LIN {X 0,Y 417.024,Z 629.46,A -85,B 0,C 180,E1 -10170,E2 -10170} C_VEL
LIN {X 0,Y 417.067,Z 628.857,A -85,B 0,C 180,E1 -10171.932,E2 -10171.932} C_VEL
LIN {X 0,Y 416.992,Z 627.097,A -85,B 0,C 180,E1 -10173.866,E2 -10173.866} C_VEL
LIN {X 0,Y 417.045,Z 624.162,A -85,B 0,C 180,E1 -10175.804,E2 -10175.804} C_VEL
LIN {X 0,Y 417.18,Z 619.979,A -85,B 0,C 180,E1 -10177.746,E2 -10177.746} C_VEL
LIN {X 0,Y 417.416,Z 614.438,A -85,B 0,C 180,E1 -10179.694,E2 -10179.694} C_VEL
LIN {X 0,Y 417.947,Z 607.397,A -85,B 0,C 180,E1 -10181.642,E2 -10181.642} C_VEL
LIN {X 0,Y 418.576,Z 598.635,A -85,B 0,C 180,E1 -10183.596,E2 -10183.596} C_VEL
LIN {X 0,Y 419.465,Z 589.337,A -85,B 0,C 180,E1 -10185.301,E2 -10185.301} C_VEL
LIN {X 0,Y 420.438,Z 579.892,A -85,B 0,C 180,E1 -10186.76,E2 -10186.76} C_VEL
LIN {X 0,Y 421.622,Z 568.231,A -85,B 0,C 180,E1 -10188.269,E2 -10188.269} C_VEL
LIN {X 0,Y 422.9,Z 555.169,A -85,B 0,C 180,E1 -10189.666,E2 -10189.666} C_VEL
LIN {X 0,Y 424.296,Z 541.374,A -85,B 0,C 180,E1 -10190.863,E2 -10190.863} C_VEL
LIN {X 0,Y 425.468,Z 527.829,A -85,B 0,C 180,E1 -10191.819,E2 -10191.819} C_VEL
LIN {X 0,Y 426.543,Z 513.678,A -85,B 0,C 180,E1 -10192.609,E2 -10192.609} C_VEL
LIN {X 0,Y 427.474,Z 498.647,A -85,B 0,C 180,E1 -10193.24,E2 -10193.24} C_VEL
LIN {X 0,Y 428.206,Z 483.459,A -85,B 0,C 180,E1 -10193.679,E2 -10193.679} C_VEL
LIN {X 0,Y 430.543,Z 350.818,A -85,B 0,C 180,E1 -10195.955,E2 -10195.955} C_VEL
LIN {X 0,Y 425.078,Z 321.561,A -85,B 0,C 180,E1 -10196.849,E2 -10196.849} C_VEL
LIN {X 0,Y 424.032,Z 316.253,A -85,B 0,C 180,E1 -10197.038,E2 -10197.038} C_VEL
LIN {X 0,Y 424.69,Z 307.553,A -85,B 0,C 180,E1 -10198.455,E2 -10198.455} C_VEL
LIN {X 0,Y 422.236,Z 296.355,A -85,B 0,C 180,E1 -10200.53,E2 -10200.53} C_VEL
LIN {X 0,Y 418.282,Z 281.009,A -85,B 0,C 180,E1 -10203.568,E2 -10203.568} C_VEL
LIN {X 0,Y 418.242,Z 281.01,A -85,B 0,C 180,E1 -10207.225,E2 -10207.225} C_VEL
LIN {X 0,Y 418.244,Z 281.002,A -85,B 0,C 180,E1 -10209.683,E2 -10209.683} C_VEL
LIN {X 0,Y 418.226,Z 281.014,A -85,B 0,C 180,E1 -10212.321,E2 -10212.321} C_VEL
LIN {X 0,Y 418.238,Z 281.01,A -85,B 0,C 180,E1 -10215.109,E2 -10215.109} C_VEL
LIN {X 0,Y 418.243,Z 281.007,A -85,B 0,C 180,E1 -10217.767,E2 -10217.767} C_VEL
LIN {X 0,Y 418.248,Z 281.012,A -85,B 0,C 180,E1 -10220.621,E2 -10220.621} C_VEL
LIN {X 0,Y 418.245,Z 281.012,A -85,B 0,C 180,E1 -10223.976,E2 -10223.976} C_VEL
LIN {X 0,Y 418.261,Z 281.003,A -85,B 0,C 180,E1 -10227.156,E2 -10227.156} C_VEL
LIN {X 0,Y 418.265,Z 281.003,A -85,B 0,C 180,E1 -10230.838,E2 -10230.838} C_VEL
LIN {X 0,Y 418.24,Z 281.008,A -85,B 0,C 180,E1 -10234.094,E2 -10234.094} C_VEL
LIN {X 0,Y 418.236,Z 281.004,A -85,B 0,C 180,E1 -10237.264,E2 -10237.264} C_VEL
LIN {X 0,Y 418.288,Z 281.002,A -85,B 0,C 180,E1 -10240.365,E2 -10240.365} C_VEL
LIN {X 0,Y 418.321,Z 281,A -85,B 0,C 180,E1 -10243.405,E2 -10243.405} C_VEL
LIN {X 0,Y 418.352,Z 280.995,A -85,B 0,C 180,E1 -10247,E2 -10247} C_VEL
LIN {X 0,Y 418.34,Z 281,A -85,B 0,C 180,E1 -10250.329,E2 -10250.329} C_VEL
LIN {X 0,Y 418.446,Z 280.978,A -85,B 0,C 180,E1 -10253.248,E2 -10253.248} C_VEL
LIN {X 0,Y 418.323,Z 281,A -85,B 0,C 180,E1 -10255.181,E2 -10255.181} C_VEL
LIN {X 0,Y 418.538,Z 280.974,A -85,B 0,C 180,E1 -10258.076,E2 -10258.076} C_VEL
LIN {X 0,Y 418.412,Z 280.986,A -85,B 0,C 180,E1 -10260.963,E2 -10260.963} C_VEL
LIN {X 0,Y 418.486,Z 280.977,A -85,B 0,C 180,E1 -10262.888,E2 -10262.888} C_VEL
LIN {X 0,Y 418.443,Z 280.98,A -85,B 0,C 180,E1 -10266.752,E2 -10266.752} C_VEL
LIN {X 0,Y 418.331,Z 280.999,A -85,B 0,C 180,E1 -10269.672,E2 -10269.672} C_VEL
LIN {X 0,Y 418.351,Z 280.996,A -85,B 0,C 180,E1 -10273,E2 -10273} C_VEL
LIN {X 0,Y 418.262,Z 281.007,A -85,B 0,C 180,E1 -10276.71,E2 -10276.71} C_VEL
LIN {X 0,Y 418.246,Z 281.012,A -85,B 0,C 180,E1 -10279.779,E2 -10279.779} C_VEL
LIN {X 0,Y 418.228,Z 281.007,A -85,B 0,C 180,E1 -10282.737,E2 -10282.737} C_VEL
LIN {X 0,Y 418.214,Z 281.01,A -85,B 0,C 180,E1 -10285.908,E2 -10285.908} C_VEL
LIN {X 0,Y 418.258,Z 280.995,A -85,B 0,C 180,E1 -10289.163,E2 -10289.163} C_VEL
LIN {X 0,Y 418.234,Z 281.009,A -85,B 0,C 180,E1 -10292.529,E2 -10292.529} C_VEL
LIN {X 0,Y 418.25,Z 281.01,A -85,B 0,C 180,E1 -10294.842,E2 -10294.842} C_VEL
LIN {X 0,Y 418.229,Z 281.008,A -85,B 0,C 180,E1 -10298.445,E2 -10298.445} C_VEL
LIN {X 0,Y 418.208,Z 281.015,A -85,B 0,C 180,E1 -10300.95,E2 -10300.95} C_VEL
LIN {X 0,Y 418.182,Z 281.017,A -85,B 0,C 180,E1 -10303.724,E2 -10303.724} C_VEL
LIN {X 0,Y 418.157,Z 281.018,A -85,B 0,C 180,E1 -10306.441,E2 -10306.441} C_VEL
LIN {X 0,Y 418.208,Z 281.018,A -85,B 0,C 180,E1 -10309.133,E2 -10309.133} C_VEL
LIN {X 0,Y 418.233,Z 281.007,A -85,B 0,C 180,E1 -10312.774,E2 -10312.774} C_VEL
LIN {X 0,Y 418.229,Z 281.009,A -85,B 0,C 180,E1 -10316.32,E2 -10316.32} C_VEL
LIN {X 0,Y 418.235,Z 281.015,A -85,B 0,C 180,E1 -10319.727,E2 -10319.727} C_VEL
LIN {X 0,Y 418.26,Z 281.079,A -85,B 0,C 180,E1 -10321.106,E2 -10321.106} C_VEL
LIN {X 0,Y 420.163,Z 288.83,A -85,B 0,C 180,E1 -10322.78,E2 -10322.78} C_VEL
LIN {X 0,Y 430.381,Z 312.246,A -85,B 0,C 180,E1 -10323.914,E2 -10323.914} C_VEL
LIN {X 0,Y 430.959,Z 315.076,A -85,B 0,C 180,E1 -10324.004,E2 -10324.004} C_VEL
LIN {X 0,Y 429.175,Z 418.752,A -85,B 0,C 180,E1 -10325.769,E2 -10325.769} C_VEL
LIN {X 0,Y 428.544,Z 454.243,A -85,B 0,C 180,E1 -10326.405,E2 -10326.405} C_VEL
LIN {X 0,Y 427.949,Z 469.526,A -85,B 0,C 180,E1 -10326.866,E2 -10326.866} C_VEL
LIN {X 0,Y 427.171,Z 484.377,A -85,B 0,C 180,E1 -10327.512,E2 -10327.512} C_VEL
LIN {X 0,Y 426.162,Z 498.888,A -85,B 0,C 180,E1 -10328.346,E2 -10328.346} C_VEL
LIN {X 0,Y 425.104,Z 512.127,A -85,B 0,C 180,E1 -10329.305,E2 -10329.305} C_VEL
LIN {X 0,Y 423.74,Z 525.582,A -85,B 0,C 180,E1 -10330.501,E2 -10330.501} C_VEL
LIN {X 0,Y 423.01,Z 533.114,A -85,B 0,C 180,E1 -10331.296,E2 -10331.296} C_VEL
LIN {X 0,Y 421.968,Z 537.683,A -85,B 0,C 180,E1 -10331.788,E2 -10331.788} C_VEL
LIN {X 0,Y 418.449,Z 544.934,A -85,B 0,C 180,E1 -10332.576,E2 -10332.576} C_VEL
LIN {X 0,Y 414.904,Z 551.847,A -85,B 0,C 180,E1 -10333.424,E2 -10333.424} C_VEL
LIN {X 0,Y 413.805,Z 555.759,A -85,B 0,C 180,E1 -10334.017,E2 -10334.017} C_VEL
LIN {X 0,Y 412.722,Z 565.22,A -85,B 0,C 180,E1 -10335.705,E2 -10335.705} C_VEL
LIN {X 0,Y 411.949,Z 573.28,A -85,B 0,C 180,E1 -10337.436,E2 -10337.436} C_VEL
LIN {X 0,Y 411.195,Z 579.932,A -85,B 0,C 180,E1 -10339.163,E2 -10339.163} C_VEL
LIN {X 0,Y 410.68,Z 586.087,A -85,B 0,C 180,E1 -10341.14,E2 -10341.14} C_VEL
LIN {X 0,Y 410.333,Z 591.474,A -85,B 0,C 180,E1 -10343.414,E2 -10343.414} C_VEL
LIN {X 0,Y 410.121,Z 594.319,A -85,B 0,C 180,E1 -10345.084,E2 -10345.084} C_VEL
LIN {X 0,Y 410.09,Z 596.618,A -85,B 0,C 180,E1 -10347.052,E2 -10347.052} C_VEL
LIN {X 0,Y 409.958,Z 597.797,A -85,B 0,C 180,E1 -10349.017,E2 -10349.017} C_VEL
LIN {X 0,Y 409.958,Z 597.814,A -85,B 0,C 180,E1 -10350.982,E2 -10350.982} C_VEL
LIN {X 0,Y 410.09,Z 596.699,A -85,B 0,C 180,E1 -10352.947,E2 -10352.947} C_VEL
LIN {X 0,Y 410.119,Z 594.463,A -85,B 0,C 180,E1 -10354.915,E2 -10354.915} C_VEL
LIN {X 0,Y 410.334,Z 591.042,A -85,B 0,C 180,E1 -10356.885,E2 -10356.885} C_VEL
LIN {X 0,Y 410.669,Z 586.356,A -85,B 0,C 180,E1 -10358.86,E2 -10358.86} C_VEL
LIN {X 0,Y 411.17,Z 580.283,A -85,B 0,C 180,E1 -10360.837,E2 -10360.837} C_VEL
LIN {X 0,Y 411.997,Z 572.627,A -85,B 0,C 180,E1 -10362.812,E2 -10362.812} C_VEL
LIN {X 0,Y 412.813,Z 564.465,A -85,B 0,C 180,E1 -10364.543,E2 -10364.543} C_VEL
LIN {X 0,Y 413.919,Z 554.624,A -85,B 0,C 180,E1 -10366.269,E2 -10366.269} C_VEL
LIN {X 0,Y 415.038,Z 544.529,A -85,B 0,C 180,E1 -10367.746,E2 -10367.746} C_VEL
LIN {X 0,Y 416.417,Z 532.505,A -85,B 0,C 180,E1 -10369.214,E2 -10369.214} C_VEL
LIN {X 0,Y 417.512,Z 521.723,A -85,B 0,C 180,E1 -10370.315,E2 -10370.315} C_VEL
LIN {X 0,Y 418.779,Z 508.898,A -85,B 0,C 180,E1 -10371.408,E2 -10371.408} C_VEL
LIN {X 0,Y 419.917,Z 494.827,A -85,B 0,C 180,E1 -10372.38,E2 -10372.38} C_VEL
LIN {X 0,Y 420.902,Z 480.644,A -85,B 0,C 180,E1 -10373.145,E2 -10373.145} C_VEL
LIN {X 0,Y 421.646,Z 465.905,A -85,B 0,C 180,E1 -10373.743,E2 -10373.743} C_VEL
LIN {X 0,Y 422.11,Z 451.888,A -85,B 0,C 180,E1 -10374.139,E2 -10374.139} C_VEL
LIN {X 0,Y 424.203,Z 342.239,A -85,B 0,C 180,E1 -10376.042,E2 -10376.042} C_VEL
LIN {X 0,Y 424.592,Z 315.602,A -85,B 0,C 180,E1 -10376.51,E2 -10376.51} C_VEL
LIN {X 0,Y 415.445,Z 294.516,A -85,B 0,C 180,E1 -10377.55,E2 -10377.55} C_VEL
LIN {X 0,Y 412.915,Z 288.768,A -85,B 0,C 180,E1 -10377.864,E2 -10377.864} C_VEL
LIN {X 0,Y 411.194,Z 281.894,A -85,B 0,C 180,E1 -10379.484,E2 -10379.484} C_VEL
LIN {X 0,Y 411.201,Z 281.889,A -85,B 0,C 180,E1 -10383.156,E2 -10383.156} C_VEL
LIN {X 0,Y 411.187,Z 281.888,A -85,B 0,C 180,E1 -10386.551,E2 -10386.551} C_VEL
LIN {X 0,Y 411.166,Z 281.892,A -85,B 0,C 180,E1 -10389.72,E2 -10389.72} C_VEL
LIN {X 0,Y 411.159,Z 281.884,A -85,B 0,C 180,E1 -10393.135,E2 -10393.135} C_VEL
LIN {X 0,Y 411.161,Z 281.892,A -85,B 0,C 180,E1 -10395.882,E2 -10395.882} C_VEL
LIN {X 0,Y 411.153,Z 281.891,A -85,B 0,C 180,E1 -10399.492,E2 -10399.492} C_VEL
LIN {X 0,Y 411.175,Z 281.889,A -85,B 0,C 180,E1 -10402.024,E2 -10402.024} C_VEL
LIN {X 0,Y 411.197,Z 281.882,A -85,B 0,C 180,E1 -10405.124,E2 -10405.124} C_VEL
LIN {X 0,Y 411.151,Z 281.893,A -85,B 0,C 180,E1 -10408.001,E2 -10408.001} C_VEL
LIN {X 0,Y 411.166,Z 281.89,A -85,B 0,C 180,E1 -10411.406,E2 -10411.406} C_VEL
LIN {X 0,Y 411.186,Z 281.89,A -85,B 0,C 180,E1 -10414.941,E2 -10414.941} C_VEL
LIN {X 0,Y 411.196,Z 281.885,A -85,B 0,C 180,E1 -10417.913,E2 -10417.913} C_VEL
LIN {X 0,Y 411.181,Z 281.883,A -85,B 0,C 180,E1 -10421.049,E2 -10421.049} C_VEL
LIN {X 0,Y 411.206,Z 281.89,A -85,B 0,C 180,E1 -10424.13,E2 -10424.13} C_VEL
LIN {X 0,Y 411.302,Z 281.872,A -85,B 0,C 180,E1 -10427.165,E2 -10427.165} C_VEL
LIN {X 0,Y 411.28,Z 281.875,A -85,B 0,C 180,E1 -10430.161,E2 -10430.161} C_VEL
LIN {X 0,Y 411.386,Z 281.863,A -85,B 0,C 180,E1 -10433.132,E2 -10433.132} C_VEL
LIN {X 0,Y 411.288,Z 281.871,A -85,B 0,C 180,E1 -10435.099,E2 -10435.099} C_VEL
LIN {X 0,Y 411.507,Z 281.851,A -85,B 0,C 180,E1 -10438.042,E2 -10438.042} C_VEL
LIN {X 0,Y 411.435,Z 281.849,A -85,B 0,C 180,E1 -10440.979,E2 -10440.979} C_VEL
LIN {X 0,Y 411.434,Z 281.857,A -85,B 0,C 180,E1 -10442.937,E2 -10442.937} C_VEL
LIN {X 0,Y 411.431,Z 281.854,A -85,B 0,C 180,E1 -10445.883,E2 -10445.883} C_VEL
LIN {X 0,Y 411.316,Z 281.872,A -85,B 0,C 180,E1 -10448.846,E2 -10448.846} C_VEL
LIN {X 0,Y 411.281,Z 281.875,A -85,B 0,C 180,E1 -10451.833,E2 -10451.833} C_VEL
LIN {X 0,Y 411.258,Z 281.874,A -85,B 0,C 180,E1 -10454.853,E2 -10454.853} C_VEL
LIN {X 0,Y 411.249,Z 281.886,A -85,B 0,C 180,E1 -10457.915,E2 -10457.915} C_VEL
LIN {X 0,Y 411.195,Z 281.888,A -85,B 0,C 180,E1 -10461.034,E2 -10461.034} C_VEL
LIN {X 0,Y 411.216,Z 281.869,A -85,B 0,C 180,E1 -10464.216,E2 -10464.216} C_VEL
LIN {X 0,Y 411.187,Z 281.885,A -85,B 0,C 180,E1 -10467.483,E2 -10467.483} C_VEL
LIN {X 0,Y 411.187,Z 281.88,A -85,B 0,C 180,E1 -10470.848,E2 -10470.848} C_VEL
LIN {X 0,Y 411.205,Z 281.888,A -85,B 0,C 180,E1 -10474.334,E2 -10474.334} C_VEL
LIN {X 0,Y 411.194,Z 281.879,A -85,B 0,C 180,E1 -10477.974,E2 -10477.974} C_VEL
LIN {X 0,Y 411.181,Z 281.889,A -85,B 0,C 180,E1 -10480.504,E2 -10480.504} C_VEL
LIN {X 0,Y 411.171,Z 281.892,A -85,B 0,C 180,E1 -10483.134,E2 -10483.134} C_VEL
LIN {X 0,Y 411.166,Z 281.894,A -85,B 0,C 180,E1 -10485.881,E2 -10485.881} C_VEL
LIN {X 0,Y 411.161,Z 281.888,A -85,B 0,C 180,E1 -10488.772,E2 -10488.772} C_VEL
LIN {X 0,Y 411.193,Z 281.89,A -85,B 0,C 180,E1 -10492.027,E2 -10492.027} C_VEL
LIN {X 0,Y 411.212,Z 281.887,A -85,B 0,C 180,E1 -10495.667,E2 -10495.667} C_VEL
LIN {X 0,Y 411.244,Z 282.008,A -85,B 0,C 180,E1 -10496.04,E2 -10496.04} C_VEL
LIN {X 0,Y 415.337,Z 297.864,A -85,B 0,C 180,E1 -10499.212,E2 -10499.212} C_VEL
LIN {X 0,Y 417.858,Z 308.784,A -85,B 0,C 180,E1 -10501.286,E2 -10501.286} C_VEL
LIN {X 0,Y 417.385,Z 316.068,A -85,B 0,C 180,E1 -10502.504,E2 -10502.504} C_VEL
LIN {X 0,Y 422.472,Z 342.049,A -85,B 0,C 180,E1 -10503.347,E2 -10503.347} C_VEL
LIN {X 0,Y 424.118,Z 352.168,A -85,B 0,C 180,E1 -10503.645,E2 -10503.645} C_VEL
LIN {X 0,Y 421.823,Z 479.15,A -85,B 0,C 180,E1 -10505.844,E2 -10505.844} C_VEL
LIN {X 0,Y 421.165,Z 494.946,A -85,B 0,C 180,E1 -10506.261,E2 -10506.261} C_VEL
LIN {X 0,Y 420.254,Z 509.586,A -85,B 0,C 180,E1 -10506.836,E2 -10506.836} C_VEL
LIN {X 0,Y 419.189,Z 523.691,A -85,B 0,C 180,E1 -10507.579,E2 -10507.579} C_VEL
LIN {X 0,Y 417.898,Z 538.017,A -85,B 0,C 180,E1 -10508.545,E2 -10508.545} C_VEL
LIN {X 0,Y 416.582,Z 551.066,A -85,B 0,C 180,E1 -10509.638,E2 -10509.638} C_VEL
LIN {X 0,Y 415.288,Z 563.121,A -85,B 0,C 180,E1 -10510.86,E2 -10510.86} C_VEL
LIN {X 0,Y 414.076,Z 574.294,A -85,B 0,C 180,E1 -10512.212,E2 -10512.212} C_VEL
LIN {X 0,Y 412.993,Z 584.581,A -85,B 0,C 180,E1 -10513.693,E2 -10513.693} C_VEL
LIN {X 0,Y 411.981,Z 594.643,A -85,B 0,C 180,E1 -10515.427,E2 -10515.427} C_VEL
LIN {X 0,Y 411.192,Z 603.004,A -85,B 0,C 180,E1 -10517.163,E2 -10517.163} C_VEL
LIN {X 0,Y 410.641,Z 610.868,A -85,B 0,C 180,E1 -10519.149,E2 -10519.149} C_VEL
LIN {X 0,Y 410.223,Z 617.126,A -85,B 0,C 180,E1 -10521.131,E2 -10521.131} C_VEL
LIN {X 0,Y 410.049,Z 621.972,A -85,B 0,C 180,E1 -10523.11,E2 -10523.11} C_VEL
LIN {X 0,Y 409.957,Z 625.523,A -85,B 0,C 180,E1 -10525.083,E2 -10525.083} C_VEL
LIN {X 0,Y 409.934,Z 627.86,A -85,B 0,C 180,E1 -10527.052,E2 -10527.052} C_VEL
LIN {X 0,Y 409.953,Z 629.036,A -85,B 0,C 180,E1 -10529.018,E2 -10529.018} C_VEL
LIN {X 0,Y 409.953,Z 629.034,A -85,B 0,C 180,E1 -10530.983,E2 -10530.983} C_VEL
LIN {X 0,Y 409.935,Z 627.851,A -85,B 0,C 180,E1 -10532.949,E2 -10532.949} C_VEL
LIN {X 0,Y 409.953,Z 625.51,A -85,B 0,C 180,E1 -10534.918,E2 -10534.918} C_VEL
LIN {X 0,Y 410.047,Z 621.961,A -85,B 0,C 180,E1 -10536.891,E2 -10536.891} C_VEL
LIN {X 0,Y 410.222,Z 617.114,A -85,B 0,C 180,E1 -10538.87,E2 -10538.87} C_VEL
LIN {X 0,Y 410.639,Z 610.843,A -85,B 0,C 180,E1 -10540.852,E2 -10540.852} C_VEL
LIN {X 0,Y 411.19,Z 602.971,A -85,B 0,C 180,E1 -10542.838,E2 -10542.838} C_VEL
LIN {X 0,Y 411.982,Z 594.608,A -85,B 0,C 180,E1 -10544.574,E2 -10544.574} C_VEL
LIN {X 0,Y 412.959,Z 584.537,A -85,B 0,C 180,E1 -10546.309,E2 -10546.309} C_VEL
LIN {X 0,Y 414.128,Z 574.249,A -85,B 0,C 180,E1 -10547.787,E2 -10547.787} C_VEL
LIN {X 0,Y 415.449,Z 561.994,A -85,B 0,C 180,E1 -10549.262,E2 -10549.262} C_VEL
LIN {X 0,Y 416.733,Z 549.7,A -85,B 0,C 180,E1 -10550.484,E2 -10550.484} C_VEL
LIN {X 0,Y 418.056,Z 536.328,A -85,B 0,C 180,E1 -10551.577,E2 -10551.577} C_VEL
LIN {X 0,Y 419.357,Z 521.576,A -85,B 0,C 180,E1 -10552.543,E2 -10552.543} C_VEL
LIN {X 0,Y 420.489,Z 506.139,A -85,B 0,C 180,E1 -10553.316,E2 -10553.316} C_VEL
LIN {X 0,Y 421.356,Z 491.063,A -85,B 0,C 180,E1 -10553.859,E2 -10553.859} C_VEL
LIN {X 0,Y 421.913,Z 475.757,A -85,B 0,C 180,E1 -10554.217,E2 -10554.217} C_VEL
LIN {X 0,Y 424.075,Z 351.155,A -85,B 0,C 180,E1 -10556.369,E2 -10556.369} C_VEL
LIN {X 0,Y 418.263,Z 320.609,A -85,B 0,C 180,E1 -10557.335,E2 -10557.335} C_VEL
LIN {X 0,Y 417.351,Z 316.082,A -85,B 0,C 180,E1 -10557.487,E2 -10557.487} C_VEL
LIN {X 0,Y 417.893,Z 309.811,A -85,B 0,C 180,E1 -10558.526,E2 -10558.526} C_VEL
LIN {X 0,Y 415.748,Z 299.421,A -85,B 0,C 180,E1 -10560.474,E2 -10560.474} C_VEL
LIN {X 0,Y 411.516,Z 283.155,A -85,B 0,C 180,E1 -10563.714,E2 -10563.714} C_VEL
LIN {X 0,Y 411.22,Z 281.889,A -85,B 0,C 180,E1 -10564,E2 -10564} C_VEL
LIN {X 0,Y 411.192,Z 281.892,A -85,B 0,C 180,E1 -10566.743,E2 -10566.743} C_VEL
LIN {X 0,Y 411.209,Z 281.878,A -85,B 0,C 180,E1 -10569.727,E2 -10569.727} C_VEL
LIN {X 0,Y 411.173,Z 281.89,A -85,B 0,C 180,E1 -10573.134,E2 -10573.134} C_VEL
LIN {X 0,Y 411.17,Z 281.887,A -85,B 0,C 180,E1 -10575.882,E2 -10575.882} C_VEL
LIN {X 0,Y 411.167,Z 281.893,A -85,B 0,C 180,E1 -10578.772,E2 -10578.772} C_VEL
LIN {X 0,Y 411.194,Z 281.889,A -85,B 0,C 180,E1 -10582.026,E2 -10582.026} C_VEL
LIN {X 0,Y 411.209,Z 281.883,A -85,B 0,C 180,E1 -10585.667,E2 -10585.667} C_VEL
LIN {X 0,Y 411.193,Z 281.885,A -85,B 0,C 180,E1 -10589.153,E2 -10589.153} C_VEL
LIN {X 0,Y 411.193,Z 281.887,A -85,B 0,C 180,E1 -10592.518,E2 -10592.518} C_VEL
LIN {X 0,Y 411.216,Z 281.886,A -85,B 0,C 180,E1 -10595.784,E2 -10595.784} C_VEL
LIN {X 0,Y 411.201,Z 281.886,A -85,B 0,C 180,E1 -10598.966,E2 -10598.966} C_VEL
LIN {X 0,Y 411.255,Z 281.882,A -85,B 0,C 180,E1 -10602.085,E2 -10602.085} C_VEL
LIN {X 0,Y 411.264,Z 281.874,A -85,B 0,C 180,E1 -10605.148,E2 -10605.148} C_VEL
LIN {X 0,Y 411.287,Z 281.874,A -85,B 0,C 180,E1 -10608.167,E2 -10608.167} C_VEL
LIN {X 0,Y 411.322,Z 281.872,A -85,B 0,C 180,E1 -10611.154,E2 -10611.154} C_VEL
LIN {X 0,Y 411.434,Z 281.861,A -85,B 0,C 180,E1 -10614.118,E2 -10614.118} C_VEL
LIN {X 0,Y 411.507,Z 281.849,A -85,B 0,C 180,E1 -10618.043,E2 -10618.043} C_VEL
LIN {X 0,Y 411.382,Z 281.861,A -85,B 0,C 180,E1 -10620.979,E2 -10620.979} C_VEL
LIN {X 0,Y 411.444,Z 281.854,A -85,B 0,C 180,E1 -10622.937,E2 -10622.937} C_VEL
LIN {X 0,Y 411.393,Z 281.859,A -85,B 0,C 180,E1 -10626.868,E2 -10626.868} C_VEL
LIN {X 0,Y 411.285,Z 281.874,A -85,B 0,C 180,E1 -10629.839,E2 -10629.839} C_VEL
LIN {X 0,Y 411.311,Z 281.874,A -85,B 0,C 180,E1 -10633.104,E2 -10633.104} C_VEL
LIN {X 0,Y 411.212,Z 281.885,A -85,B 0,C 180,E1 -10636.891,E2 -10636.891} C_VEL
LIN {X 0,Y 411.208,Z 281.888,A -85,B 0,C 180,E1 -10639.988,E2 -10639.988} C_VEL
LIN {X 0,Y 411.188,Z 281.885,A -85,B 0,C 180,E1 -10643.149,E2 -10643.149} C_VEL
LIN {X 0,Y 411.167,Z 281.885,A -85,B 0,C 180,E1 -10646.386,E2 -10646.386} C_VEL
LIN {X 0,Y 411.196,Z 281.883,A -85,B 0,C 180,E1 -10649.713,E2 -10649.713} C_VEL
LIN {X 0,Y 411.206,Z 281.886,A -85,B 0,C 180,E1 -10653.156,E2 -10653.156} C_VEL
LIN {X 0,Y 411.19,Z 281.885,A -85,B 0,C 180,E1 -10656.551,E2 -10656.551} C_VEL
LIN {X 0,Y 411.166,Z 281.893,A -85,B 0,C 180,E1 -10659.719,E2 -10659.719} C_VEL
LIN {X 0,Y 411.12,Z 281.9,A -85,B 0,C 180,E1 -10663.141,E2 -10663.141} C_VEL
LIN {X 0,Y 411.111,Z 281.896,A -85,B 0,C 180,E1 -10665.889,E2 -10665.889} C_VEL
LIN {X 0,Y 411.158,Z 281.895,A -85,B 0,C 180,E1 -10669.492,E2 -10669.492} C_VEL
LIN {X 0,Y 411.179,Z 281.888,A -85,B 0,C 180,E1 -10672.024,E2 -10672.024} C_VEL
LIN {X 0,Y 411.201,Z 281.887,A -85,B 0,C 180,E1 -10675.124,E2 -10675.124} C_VEL
LIN {X 0,Y 411.155,Z 281.891,A -85,B 0,C 180,E1 -10678.001,E2 -10678.001} C_VEL
LIN {X 0,Y 411.218,Z 281.932,A -85,B 0,C 180,E1 -10680.683,E2 -10680.683} C_VEL
LIN {X 0,Y 412.926,Z 288.883,A -85,B 0,C 180,E1 -10682.257,E2 -10682.257} C_VEL
LIN {X 0,Y 423.835,Z 313.789,A -85,B 0,C 180,E1 -10683.503,E2 -10683.503} C_VEL
LIN {X 0,Y 424.541,Z 315.615,A -85,B 0,C 180,E1 -10683.585,E2 -10683.585} C_VEL
LIN {X 0,Y 422.796,Z 417.26,A -85,B 0,C 180,E1 -10685.346,E2 -10685.346} C_VEL
LIN {X 0,Y 422.061,Z 454.53,A -85,B 0,C 180,E1 -10686.02,E2 -10686.02} C_VEL
LIN {X 0,Y 421.457,Z 469.531,A -85,B 0,C 180,E1 -10686.477,E2 -10686.477} C_VEL
LIN {X 0,Y 420.629,Z 484.849,A -85,B 0,C 180,E1 -10687.154,E2 -10687.154} C_VEL
LIN {X 0,Y 419.586,Z 499.164,A -85,B 0,C 180,E1 -10687.989,E2 -10687.989} C_VEL
LIN {X 0,Y 418.456,Z 512.403,A -85,B 0,C 180,E1 -10688.961,E2 -10688.961} C_VEL
LIN {X 0,Y 417.045,Z 525.857,A -85,B 0,C 180,E1 -10690.175,E2 -10690.175} C_VEL
LIN {X 0,Y 415.803,Z 538.049,A -85,B 0,C 180,E1 -10691.523,E2 -10691.523} C_VEL
LIN {X 0,Y 414.582,Z 549.15,A -85,B 0,C 180,E1 -10692.996,E2 -10692.996} C_VEL
LIN {X 0,Y 413.805,Z 555.759,A -85,B 0,C 180,E1 -10694.017,E2 -10694.017} C_VEL
LIN {X 0,Y 412.723,Z 559.602,A -85,B 0,C 180,E1 -10694.631,E2 -10694.631} C_VEL
LIN {X 0,Y 406.401,Z 570.041,A -85,B 0,C 180,E1 -10696.448,E2 -10696.448} C_VEL
LIN {X 0,Y 405.096,Z 573.179,A -85,B 0,C 180,E1 -10697.13,E2 -10697.13} C_VEL
LIN {X 0,Y 404.938,Z 574.161,A -85,B 0,C 180,E1 -10697.37,E2 -10697.37} C_VEL
LIN {X 0,Y 404.046,Z 581.873,A -85,B 0,C 180,E1 -10699.476,E2 -10699.476} C_VEL
LIN {X 0,Y 403.538,Z 587.676,A -85,B 0,C 180,E1 -10701.486,E2 -10701.486} C_VEL
LIN {X 0,Y 403.271,Z 591.946,A -85,B 0,C 180,E1 -10703.398,E2 -10703.398} C_VEL
LIN {X 0,Y 403.06,Z 594.589,A -85,B 0,C 180,E1 -10704.998,E2 -10704.998} C_VEL
LIN {X 0,Y 402.992,Z 596.889,A -85,B 0,C 180,E1 -10707.001,E2 -10707.001} C_VEL
LIN {X 0,Y 402.884,Z 598.067,A -85,B 0,C 180,E1 -10709,E2 -10709} C_VEL
LIN {X 0,Y 402.884,Z 598.083,A -85,B 0,C 180,E1 -10710.999,E2 -10710.999} C_VEL
LIN {X 0,Y 402.992,Z 596.969,A -85,B 0,C 180,E1 -10712.999,E2 -10712.999} C_VEL
LIN {X 0,Y 403.058,Z 594.733,A -85,B 0,C 180,E1 -10715.001,E2 -10715.001} C_VEL
LIN {X 0,Y 403.272,Z 591.312,A -85,B 0,C 180,E1 -10717.007,E2 -10717.007} C_VEL
LIN {X 0,Y 403.649,Z 586.626,A -85,B 0,C 180,E1 -10719.015,E2 -10719.015} C_VEL
LIN {X 0,Y 404.164,Z 580.553,A -85,B 0,C 180,E1 -10721.027,E2 -10721.027} C_VEL
LIN {X 0,Y 405.048,Z 572.897,A -85,B 0,C 180,E1 -10723.036,E2 -10723.036} C_VEL
LIN {X 0,Y 405.91,Z 564.734,A -85,B 0,C 180,E1 -10724.796,E2 -10724.796} C_VEL
LIN {X 0,Y 407.094,Z 554.892,A -85,B 0,C 180,E1 -10726.55,E2 -10726.55} C_VEL
LIN {X 0,Y 408.256,Z 544.797,A -85,B 0,C 180,E1 -10728.051,E2 -10728.051} C_VEL
LIN {X 0,Y 409.719,Z 532.772,A -85,B 0,C 180,E1 -10729.54,E2 -10729.54} C_VEL
LIN {X 0,Y 410.875,Z 521.988,A -85,B 0,C 180,E1 -10730.658,E2 -10730.658} C_VEL
LIN {X 0,Y 412.174,Z 509.162,A -85,B 0,C 180,E1 -10731.768,E2 -10731.768} C_VEL
LIN {X 0,Y 413.366,Z 495.09,A -85,B 0,C 180,E1 -10732.755,E2 -10732.755} C_VEL
LIN {X 0,Y 414.421,Z 480.226,A -85,B 0,C 180,E1 -10733.564,E2 -10733.564} C_VEL
LIN {X 0,Y 415.198,Z 465.249,A -85,B 0,C 180,E1 -10734.168,E2 -10734.168} C_VEL
LIN {X 0,Y 415.755,Z 450.631,A -85,B 0,C 180,E1 -10734.565,E2 -10734.565} C_VEL
LIN {X 0,Y 417.913,Z 337.717,A -85,B 0,C 180,E1 -10736.554,E2 -10736.554} C_VEL
LIN {X 0,Y 418.174,Z 317.36,A -85,B 0,C 180,E1 -10736.921,E2 -10736.921} C_VEL
LIN {X 0,Y 408.769,Z 295.62,A -85,B 0,C 180,E1 -10738.023,E2 -10738.023} C_VEL
LIN {X 0,Y 405.704,Z 288.989,A -85,B 0,C 180,E1 -10738.42,E2 -10738.42} C_VEL
LIN {X 0,Y 404.15,Z 282.773,A -85,B 0,C 180,E1 -10739.895,E2 -10739.895} C_VEL
LIN {X 0,Y 404.165,Z 282.766,A -85,B 0,C 180,E1 -10743.418,E2 -10743.418} C_VEL
LIN {X 0,Y 404.132,Z 282.765,A -85,B 0,C 180,E1 -10746.247,E2 -10746.247} C_VEL
LIN {X 0,Y 404.131,Z 282.772,A -85,B 0,C 180,E1 -10748.759,E2 -10748.759} C_VEL
LIN {X 0,Y 404.103,Z 282.771,A -85,B 0,C 180,E1 -10751.596,E2 -10751.596} C_VEL
LIN {X 0,Y 404.141,Z 282.764,A -85,B 0,C 180,E1 -10754.521,E2 -10754.521} C_VEL
LIN {X 0,Y 404.117,Z 282.756,A -85,B 0,C 180,E1 -10757.293,E2 -10757.293} C_VEL
LIN {X 0,Y 404.131,Z 282.766,A -85,B 0,C 180,E1 -10759.951,E2 -10759.951} C_VEL
LIN {X 0,Y 404.127,Z 282.749,A -85,B 0,C 180,E1 -10763.126,E2 -10763.126} C_VEL
LIN {X 0,Y 404.133,Z 282.766,A -85,B 0,C 180,E1 -10766.187,E2 -10766.187} C_VEL
LIN {X 0,Y 404.137,Z 282.765,A -85,B 0,C 180,E1 -10769.714,E2 -10769.714} C_VEL
LIN {X 0,Y 404.1,Z 282.771,A -85,B 0,C 180,E1 -10773.116,E2 -10773.116} C_VEL
LIN {X 0,Y 404.144,Z 282.764,A -85,B 0,C 180,E1 -10776.424,E2 -10776.424} C_VEL
LIN {X 0,Y 404.148,Z 282.766,A -85,B 0,C 180,E1 -10779.89,E2 -10779.89} C_VEL
LIN {X 0,Y 404.153,Z 282.766,A -85,B 0,C 180,E1 -10783.022,E2 -10783.022} C_VEL
LIN {X 0,Y 404.282,Z 282.748,A -85,B 0,C 180,E1 -10786.939,E2 -10786.939} C_VEL
LIN {X 0,Y 404.247,Z 282.753,A -85,B 0,C 180,E1 -10789.988,E2 -10789.988} C_VEL
LIN {X 0,Y 404.337,Z 282.742,A -85,B 0,C 180,E1 -10793.011,E2 -10793.011} C_VEL
LIN {X 0,Y 404.258,Z 282.746,A -85,B 0,C 180,E1 -10795.013,E2 -10795.013} C_VEL
LIN {X 0,Y 404.476,Z 282.726,A -85,B 0,C 180,E1 -10798.008,E2 -10798.008} C_VEL
LIN {X 0,Y 404.4,Z 282.725,A -85,B 0,C 180,E1 -10800.996,E2 -10800.996} C_VEL
LIN {X 0,Y 404.393,Z 282.734,A -85,B 0,C 180,E1 -10802.988,E2 -10802.988} C_VEL
LIN {X 0,Y 404.379,Z 282.732,A -85,B 0,C 180,E1 -10805.985,E2 -10805.985} C_VEL
LIN {X 0,Y 404.263,Z 282.75,A -85,B 0,C 180,E1 -10809.002,E2 -10809.002} C_VEL
LIN {X 0,Y 404.254,Z 282.753,A -85,B 0,C 180,E1 -10812.041,E2 -10812.041} C_VEL
LIN {X 0,Y 404.204,Z 282.752,A -85,B 0,C 180,E1 -10815.118,E2 -10815.118} C_VEL
LIN {X 0,Y 404.206,Z 282.759,A -85,B 0,C 180,E1 -10818.238,E2 -10818.238} C_VEL
LIN {X 0,Y 404.137,Z 282.769,A -85,B 0,C 180,E1 -10821.419,E2 -10821.419} C_VEL
LIN {X 0,Y 404.165,Z 282.744,A -85,B 0,C 180,E1 -10824.666,E2 -10824.666} C_VEL
LIN {X 0,Y 404.129,Z 282.771,A -85,B 0,C 180,E1 -10828.005,E2 -10828.005} C_VEL
LIN {X 0,Y 404.142,Z 282.76,A -85,B 0,C 180,E1 -10830.285,E2 -10830.285} C_VEL
LIN {X 0,Y 404.143,Z 282.764,A -85,B 0,C 180,E1 -10833.812,E2 -10833.812} C_VEL
LIN {X 0,Y 404.135,Z 282.759,A -85,B 0,C 180,E1 -10836.875,E2 -10836.875} C_VEL
LIN {X 0,Y 404.146,Z 282.768,A -85,B 0,C 180,E1 -10840.08,E2 -10840.08} C_VEL
LIN {X 0,Y 404.151,Z 282.766,A -85,B 0,C 180,E1 -10843.084,E2 -10843.084} C_VEL
LIN {X 0,Y 404.146,Z 282.767,A -85,B 0,C 180,E1 -10845.926,E2 -10845.926} C_VEL
LIN {X 0,Y 404.116,Z 282.766,A -85,B 0,C 180,E1 -10848.635,E2 -10848.635} C_VEL
LIN {X 0,Y 404.152,Z 282.767,A -85,B 0,C 180,E1 -10851.492,E2 -10851.492} C_VEL
LIN {X 0,Y 404.162,Z 282.769,A -85,B 0,C 180,E1 -10855.286,E2 -10855.286} C_VEL
LIN {X 0,Y 404.2,Z 282.924,A -85,B 0,C 180,E1 -10855.592,E2 -10855.592} C_VEL
LIN {X 0,Y 408.033,Z 297.686,A -85,B 0,C 180,E1 -10858.621,E2 -10858.621} C_VEL
LIN {X 0,Y 410.922,Z 309.971,A -85,B 0,C 180,E1 -10861.014,E2 -10861.014} C_VEL
LIN {X 0,Y 410.924,Z 313.697,A -85,B 0,C 180,E1 -10861.666,E2 -10861.666} C_VEL
LIN {X 0,Y 410.734,Z 315.723,A -85,B 0,C 180,E1 -10862.007,E2 -10862.007} C_VEL
LIN {X 0,Y 415.04,Z 337.414,A -85,B 0,C 180,E1 -10862.748,E2 -10862.748} C_VEL
LIN {X 0,Y 417.76,Z 353.1,A -85,B 0,C 180,E1 -10863.234,E2 -10863.234} C_VEL
LIN {X 0,Y 415.343,Z 478.895,A -85,B 0,C 180,E1 -10865.442,E2 -10865.442} C_VEL
LIN {X 0,Y 414.659,Z 494.685,A -85,B 0,C 180,E1 -10865.865,E2 -10865.865} C_VEL
LIN {X 0,Y 413.659,Z 510.084,A -85,B 0,C 180,E1 -10866.483,E2 -10866.483} C_VEL
LIN {X 0,Y 412.619,Z 523.426,A -85,B 0,C 180,E1 -10867.202,E2 -10867.202} C_VEL
LIN {X 0,Y 411.259,Z 537.749,A -85,B 0,C 180,E1 -10868.181,E2 -10868.181} C_VEL
LIN {X 0,Y 409.879,Z 550.797,A -85,B 0,C 180,E1 -10869.29,E2 -10869.29} C_VEL
LIN {X 0,Y 408.392,Z 563.927,A -85,B 0,C 180,E1 -10870.654,E2 -10870.654} C_VEL
LIN {X 0,Y 407.06,Z 575.819,A -85,B 0,C 180,E1 -10872.155,E2 -10872.155} C_VEL
LIN {X 0,Y 405.926,Z 585.832,A -85,B 0,C 180,E1 -10873.66,E2 -10873.66} C_VEL
LIN {X 0,Y 404.905,Z 595.636,A -85,B 0,C 180,E1 -10875.424,E2 -10875.424} C_VEL
LIN {X 0,Y 404.131,Z 603.823,A -85,B 0,C 180,E1 -10877.19,E2 -10877.19} C_VEL
LIN {X 0,Y 403.594,Z 610.596,A -85,B 0,C 180,E1 -10878.957,E2 -10878.957} C_VEL
LIN {X 0,Y 403.151,Z 616.854,A -85,B 0,C 180,E1 -10880.974,E2 -10880.974} C_VEL
LIN {X 0,Y 402.97,Z 621.701,A -85,B 0,C 180,E1 -10882.988,E2 -10882.988} C_VEL
LIN {X 0,Y 402.87,Z 625.252,A -85,B 0,C 180,E1 -10884.997,E2 -10884.997} C_VEL
LIN {X 0,Y 402.833,Z 627.589,A -85,B 0,C 180,E1 -10887,E2 -10887} C_VEL
LIN {X 0,Y 402.879,Z 628.766,A -85,B 0,C 180,E1 -10889.001,E2 -10889.001} C_VEL
LIN {X 0,Y 402.879,Z 628.765,A -85,B 0,C 180,E1 -10891,E2 -10891} C_VEL
LIN {X 0,Y 402.833,Z 627.58,A -85,B 0,C 180,E1 -10893.001,E2 -10893.001} C_VEL
LIN {X 0,Y 402.867,Z 625.239,A -85,B 0,C 180,E1 -10895.004,E2 -10895.004} C_VEL
LIN {X 0,Y 402.968,Z 621.689,A -85,B 0,C 180,E1 -10897.013,E2 -10897.013} C_VEL
LIN {X 0,Y 403.149,Z 616.84,A -85,B 0,C 180,E1 -10899.027,E2 -10899.027} C_VEL
LIN {X 0,Y 403.591,Z 610.569,A -85,B 0,C 180,E1 -10901.044,E2 -10901.044} C_VEL
LIN {X 0,Y 404.159,Z 602.694,A -85,B 0,C 180,E1 -10903.066,E2 -10903.066} C_VEL
LIN {X 0,Y 405.023,Z 594.332,A -85,B 0,C 180,E1 -10904.83,E2 -10904.83} C_VEL
LIN {X 0,Y 406.094,Z 584.262,A -85,B 0,C 180,E1 -10906.593,E2 -10906.593} C_VEL
LIN {X 0,Y 407.285,Z 573.972,A -85,B 0,C 180,E1 -10908.096,E2 -10908.096} C_VEL
LIN {X 0,Y 408.696,Z 561.718,A -85,B 0,C 180,E1 -10909.593,E2 -10909.593} C_VEL
LIN {X 0,Y 410.191,Z 548.082,A -85,B 0,C 180,E1 -10910.957,E2 -10910.957} C_VEL
LIN {X 0,Y 411.563,Z 534.417,A -85,B 0,C 180,E1 -10912.067,E2 -10912.067} C_VEL
LIN {X 0,Y 412.882,Z 520.27,A -85,B 0,C 180,E1 -10912.982,E2 -10912.982} C_VEL
LIN {X 0,Y 414.008,Z 505.056,A -85,B 0,C 180,E1 -10913.74,E2 -10913.74} C_VEL
LIN {X 0,Y 414.91,Z 489.755,A -85,B 0,C 180,E1 -10914.287,E2 -10914.287} C_VEL
LIN {X 0,Y 415.48,Z 473.768,A -85,B 0,C 180,E1 -10914.65,E2 -10914.65} C_VEL
LIN {X 0,Y 417.712,Z 352.266,A -85,B 0,C 180,E1 -10916.776,E2 -10916.776} C_VEL
LIN {X 0,Y 411.84,Z 321.187,A -85,B 0,C 180,E1 -10917.781,E2 -10917.781} C_VEL
LIN {X 0,Y 410.739,Z 315.67,A -85,B 0,C 180,E1 -10917.992,E2 -10917.992} C_VEL
LIN {X 0,Y 411.074,Z 311.004,A -85,B 0,C 180,E1 -10918.785,E2 -10918.785} C_VEL
LIN {X 0,Y 408.837,Z 300.847,A -85,B 0,C 180,E1 -10920.739,E2 -10920.739} C_VEL
LIN {X 0,Y 404.648,Z 284.481,A -85,B 0,C 180,E1 -10924.065,E2 -10924.065} C_VEL
LIN {X 0,Y 404.167,Z 282.767,A -85,B 0,C 180,E1 -10924.45,E2 -10924.45} C_VEL
LIN {X 0,Y 404.142,Z 282.766,A -85,B 0,C 180,E1 -10927.493,E2 -10927.493} C_VEL
LIN {X 0,Y 404.15,Z 282.759,A -85,B 0,C 180,E1 -10930.081,E2 -10930.081} C_VEL
LIN {X 0,Y 404.152,Z 282.765,A -85,B 0,C 180,E1 -10933.084,E2 -10933.084} C_VEL
LIN {X 0,Y 404.15,Z 282.76,A -85,B 0,C 180,E1 -10935.926,E2 -10935.926} C_VEL
LIN {X 0,Y 404.122,Z 282.772,A -85,B 0,C 180,E1 -10938.635,E2 -10938.635} C_VEL
LIN {X 0,Y 404.153,Z 282.765,A -85,B 0,C 180,E1 -10941.493,E2 -10941.493} C_VEL
LIN {X 0,Y 404.188,Z 282.757,A -85,B 0,C 180,E1 -10944.984,E2 -10944.984} C_VEL
LIN {X 0,Y 404.146,Z 282.766,A -85,B 0,C 180,E1 -10948.554,E2 -10948.554} C_VEL
LIN {X 0,Y 404.161,Z 282.76,A -85,B 0,C 180,E1 -10950.863,E2 -10950.863} C_VEL
LIN {X 0,Y 404.154,Z 282.763,A -85,B 0,C 180,E1 -10954.232,E2 -10954.232} C_VEL
LIN {X 0,Y 404.172,Z 282.757,A -85,B 0,C 180,E1 -10957.508,E2 -10957.508} C_VEL
LIN {X 0,Y 404.169,Z 282.758,A -85,B 0,C 180,E1 -10960.708,E2 -10960.708} C_VEL
LIN {X 0,Y 404.226,Z 282.758,A -85,B 0,C 180,E1 -10963.848,E2 -10963.848} C_VEL
LIN {X 0,Y 404.288,Z 282.748,A -85,B 0,C 180,E1 -10966.939,E2 -10966.939} C_VEL
LIN {X 0,Y 404.259,Z 282.753,A -85,B 0,C 180,E1 -10969.988,E2 -10969.988} C_VEL
LIN {X 0,Y 404.346,Z 282.734,A -85,B 0,C 180,E1 -10973.012,E2 -10973.012} C_VEL
LIN {X 0,Y 404.266,Z 282.75,A -85,B 0,C 180,E1 -10975.013,E2 -10975.013} C_VEL
LIN {X 0,Y 404.476,Z 282.724,A -85,B 0,C 180,E1 -10978.009,E2 -10978.009} C_VEL
LIN {X 0,Y 404.352,Z 282.737,A -85,B 0,C 180,E1 -10980.996,E2 -10980.996} C_VEL
LIN {X 0,Y 404.403,Z 282.732,A -85,B 0,C 180,E1 -10982.989,E2 -10982.989} C_VEL
LIN {X 0,Y 404.343,Z 282.737,A -85,B 0,C 180,E1 -10986.989,E2 -10986.989} C_VEL
LIN {X 0,Y 404.253,Z 282.749,A -85,B 0,C 180,E1 -10990.012,E2 -10990.012} C_VEL
LIN {X 0,Y 404.272,Z 282.752,A -85,B 0,C 180,E1 -10993.211,E2 -10993.211} C_VEL
LIN {X 0,Y 404.159,Z 282.764,A -85,B 0,C 180,E1 -10996.978,E2 -10996.978} C_VEL
LIN {X 0,Y 404.155,Z 282.765,A -85,B 0,C 180,E1 -11000.352,E2 -11000.352} C_VEL
LIN {X 0,Y 404.15,Z 282.766,A -85,B 0,C 180,E1 -11003.576,E2 -11003.576} C_VEL
LIN {X 0,Y 404.101,Z 282.764,A -85,B 0,C 180,E1 -11006.884,E2 -11006.884} C_VEL
LIN {X 0,Y 404.142,Z 282.765,A -85,B 0,C 180,E1 -11010.286,E2 -11010.286} C_VEL
LIN {X 0,Y 404.139,Z 282.769,A -85,B 0,C 180,E1 -11013.813,E2 -11013.813} C_VEL
LIN {X 0,Y 404.132,Z 282.766,A -85,B 0,C 180,E1 -11016.873,E2 -11016.873} C_VEL
LIN {X 0,Y 404.12,Z 282.768,A -85,B 0,C 180,E1 -11020.074,E2 -11020.074} C_VEL
LIN {X 0,Y 404.079,Z 282.777,A -85,B 0,C 180,E1 -11023.072,E2 -11023.072} C_VEL
LIN {X 0,Y 404.072,Z 282.773,A -85,B 0,C 180,E1 -11025.915,E2 -11025.915} C_VEL
LIN {X 0,Y 404.088,Z 282.772,A -85,B 0,C 180,E1 -11028.63,E2 -11028.63} C_VEL
LIN {X 0,Y 404.135,Z 282.769,A -85,B 0,C 180,E1 -11031.496,E2 -11031.496} C_VEL
LIN {X 0,Y 404.173,Z 282.764,A -85,B 0,C 180,E1 -11034.982,E2 -11034.982} C_VEL
LIN {X 0,Y 404.132,Z 282.765,A -85,B 0,C 180,E1 -11038.444,E2 -11038.444} C_VEL
LIN {X 0,Y 404.162,Z 282.828,A -85,B 0,C 180,E1 -11040.249,E2 -11040.249} C_VEL
LIN {X 0,Y 405.748,Z 289.113,A -85,B 0,C 180,E1 -11041.711,E2 -11041.711} C_VEL
LIN {X 0,Y 416.487,Z 313.281,A -85,B 0,C 180,E1 -11042.982,E2 -11042.982} C_VEL
LIN {X 0,Y 418.165,Z 317.327,A -85,B 0,C 180,E1 -11043.177,E2 -11043.177} C_VEL
LIN {X 0,Y 416.451,Z 415.768,A -85,B 0,C 180,E1 -11044.912,E2 -11044.912} C_VEL
LIN {X 0,Y 415.621,Z 453.631,A -85,B 0,C 180,E1 -11045.592,E2 -11045.592} C_VEL
LIN {X 0,Y 415.029,Z 468.788,A -85,B 0,C 180,E1 -11046.048,E2 -11046.048} C_VEL
LIN {X 0,Y 414.227,Z 483.93,A -85,B 0,C 180,E1 -11046.712,E2 -11046.712} C_VEL
LIN {X 0,Y 413.19,Z 497.554,A -85,B 0,C 180,E1 -11047.498,E2 -11047.498} C_VEL
LIN {X 0,Y 411.979,Z 511.121,A -85,B 0,C 180,E1 -11048.483,E2 -11048.483} C_VEL
LIN {X 0,Y 410.64,Z 523.596,A -85,B 0,C 180,E1 -11049.591,E2 -11049.591} C_VEL
LIN {X 0,Y 409.475,Z 534.312,A -85,B 0,C 180,E1 -11050.733,E2 -11050.733} C_VEL
LIN {X 0,Y 408.141,Z 545.894,A -85,B 0,C 180,E1 -11052.202,E2 -11052.202} C_VEL
LIN {X 0,Y 406.886,Z 556.577,A -85,B 0,C 180,E1 -11053.833,E2 -11053.833} C_VEL
LIN {X 0,Y 405.809,Z 565.494,A -85,B 0,C 180,E1 -11055.456,E2 -11055.456} C_VEL
LIN {X 0,Y 404.938,Z 574.161,A -85,B 0,C 180,E1 -11057.37,E2 -11057.37} C_VEL
LIN {X 0,Y 404.035,Z 577.11,A -85,B 0,C 180,E1 -11058.09,E2 -11058.09} C_VEL
LIN {X 0,Y 400.713,Z 581.598,A -85,B 0,C 180,E1 -11059.257,E2 -11059.257} C_VEL
LIN {X 0,Y 397.396,Z 585.604,A -85,B 0,C 180,E1 -11060.471,E2 -11060.471} C_VEL
LIN {X 0,Y 396.517,Z 587.745,A -85,B 0,C 180,E1 -11061.255,E2 -11061.255} C_VEL
LIN {X 0,Y 396.201,Z 592.415,A -85,B 0,C 180,E1 -11063.392,E2 -11063.392} C_VEL
LIN {X 0,Y 396.002,Z 594.86,A -85,B 0,C 180,E1 -11064.909,E2 -11064.909} C_VEL
LIN {X 0,Y 395.895,Z 597.16,A -85,B 0,C 180,E1 -11066.947,E2 -11066.947} C_VEL
LIN {X 0,Y 395.813,Z 598.337,A -85,B 0,C 180,E1 -11068.982,E2 -11068.982} C_VEL
LIN {X 0,Y 395.813,Z 598.352,A -85,B 0,C 180,E1 -11071.017,E2 -11071.017} C_VEL
LIN {X 0,Y 395.894,Z 597.24,A -85,B 0,C 180,E1 -11073.052,E2 -11073.052} C_VEL
LIN {X 0,Y 395.999,Z 595.002,A -85,B 0,C 180,E1 -11075.091,E2 -11075.091} C_VEL
LIN {X 0,Y 396.208,Z 591.582,A -85,B 0,C 180,E1 -11077.132,E2 -11077.132} C_VEL
LIN {X 0,Y 396.602,Z 586.896,A -85,B 0,C 180,E1 -11079.177,E2 -11079.177} C_VEL
LIN {X 0,Y 397.168,Z 580.823,A -85,B 0,C 180,E1 -11081.224,E2 -11081.224} C_VEL
LIN {X 0,Y 397.985,Z 574.214,A -85,B 0,C 180,E1 -11083.011,E2 -11083.011} C_VEL
LIN {X 0,Y 398.865,Z 566.231,A -85,B 0,C 180,E1 -11084.802,E2 -11084.802} C_VEL
LIN {X 0,Y 400.06,Z 556.642,A -85,B 0,C 180,E1 -11086.586,E2 -11086.586} C_VEL
LIN {X 0,Y 401.29,Z 546.834,A -85,B 0,C 180,E1 -11088.111,E2 -11088.111} C_VEL
LIN {X 0,Y 402.72,Z 535.166,A -85,B 0,C 180,E1 -11089.629,E2 -11089.629} C_VEL
LIN {X 0,Y 404.068,Z 523.538,A -85,B 0,C 180,E1 -11090.889,E2 -11090.889} C_VEL
LIN {X 0,Y 405.448,Z 511,A -85,B 0,C 180,E1 -11092.014,E2 -11092.014} C_VEL
LIN {X 0,Y 406.694,Z 497.332,A -85,B 0,C 180,E1 -11093.015,E2 -11093.015} C_VEL
LIN {X 0,Y 407.758,Z 483.485,A -85,B 0,C 180,E1 -11093.816,E2 -11093.816} C_VEL
LIN {X 0,Y 408.643,Z 468.243,A -85,B 0,C 180,E1 -11094.479,E2 -11094.479} C_VEL
LIN {X 0,Y 409.186,Z 453.862,A -85,B 0,C 180,E1 -11094.919,E2 -11094.919} C_VEL
LIN {X 0,Y 411.172,Z 359.488,A -85,B 0,C 180,E1 -11096.612,E2 -11096.612} C_VEL
LIN {X 0,Y 411.916,Z 319.365,A -85,B 0,C 180,E1 -11097.33,E2 -11097.33} C_VEL
LIN {X 0,Y 402.769,Z 298.429,A -85,B 0,C 180,E1 -11098.427,E2 -11098.427} C_VEL
LIN {X 0,Y 398.529,Z 289.314,A -85,B 0,C 180,E1 -11098.974,E2 -11098.974} C_VEL
LIN {X 0,Y 397.094,Z 283.648,A -85,B 0,C 180,E1 -11100.326,E2 -11100.326} C_VEL
LIN {X 0,Y 397.095,Z 283.648,A -85,B 0,C 180,E1 -11103.713,E2 -11103.713} C_VEL
LIN {X 0,Y 397.086,Z 283.652,A -85,B 0,C 180,E1 -11107.207,E2 -11107.207} C_VEL
LIN {X 0,Y 397.053,Z 283.651,A -85,B 0,C 180,E1 -11110.437,E2 -11110.437} C_VEL
LIN {X 0,Y 397.084,Z 283.638,A -85,B 0,C 180,E1 -11113.65,E2 -11113.65} C_VEL
LIN {X 0,Y 397.088,Z 283.641,A -85,B 0,C 180,E1 -11116.523,E2 -11116.523} C_VEL
LIN {X 0,Y 397.082,Z 283.648,A -85,B 0,C 180,E1 -11120.419,E2 -11120.419} C_VEL
LIN {X 0,Y 397.089,Z 283.627,A -85,B 0,C 180,E1 -11123.004,E2 -11123.004} C_VEL
LIN {X 0,Y 397.108,Z 283.647,A -85,B 0,C 180,E1 -11126.726,E2 -11126.726} C_VEL
LIN {X 0,Y 397.111,Z 283.643,A -85,B 0,C 180,E1 -11130.295,E2 -11130.295} C_VEL
LIN {X 0,Y 397.072,Z 283.645,A -85,B 0,C 180,E1 -11133.737,E2 -11133.737} C_VEL
LIN {X 0,Y 397.097,Z 283.641,A -85,B 0,C 180,E1 -11137.085,E2 -11137.085} C_VEL
LIN {X 0,Y 397.094,Z 283.643,A -85,B 0,C 180,E1 -11140.35,E2 -11140.35} C_VEL
LIN {X 0,Y 397.118,Z 283.641,A -85,B 0,C 180,E1 -11143.551,E2 -11143.551} C_VEL
LIN {X 0,Y 397.228,Z 283.626,A -85,B 0,C 180,E1 -11146.703,E2 -11146.703} C_VEL
LIN {X 0,Y 397.208,Z 283.63,A -85,B 0,C 180,E1 -11149.809,E2 -11149.809} C_VEL
LIN {X 0,Y 397.29,Z 283.621,A -85,B 0,C 180,E1 -11152.887,E2 -11152.887} C_VEL
LIN {X 0,Y 397.229,Z 283.622,A -85,B 0,C 180,E1 -11154.925,E2 -11154.925} C_VEL
LIN {X 0,Y 397.444,Z 283.602,A -85,B 0,C 180,E1 -11157.973,E2 -11157.973} C_VEL
LIN {X 0,Y 397.44,Z 283.597,A -85,B 0,C 180,E1 -11162.027,E2 -11162.027} C_VEL
LIN {X 0,Y 397.33,Z 283.61,A -85,B 0,C 180,E1 -11166.092,E2 -11166.092} C_VEL
LIN {X 0,Y 397.233,Z 283.626,A -85,B 0,C 180,E1 -11169.162,E2 -11169.162} C_VEL
LIN {X 0,Y 397.217,Z 283.633,A -85,B 0,C 180,E1 -11172.258,E2 -11172.258} C_VEL
LIN {X 0,Y 397.177,Z 283.628,A -85,B 0,C 180,E1 -11175.392,E2 -11175.392} C_VEL
LIN {X 0,Y 397.159,Z 283.634,A -85,B 0,C 180,E1 -11178.573,E2 -11178.573} C_VEL
LIN {X 0,Y 397.095,Z 283.65,A -85,B 0,C 180,E1 -11181.818,E2 -11181.818} C_VEL
LIN {X 0,Y 397.122,Z 283.618,A -85,B 0,C 180,E1 -11185.134,E2 -11185.134} C_VEL
LIN {X 0,Y 397.077,Z 283.647,A -85,B 0,C 180,E1 -11188.547,E2 -11188.547} C_VEL
LIN {X 0,Y 397.079,Z 283.63,A -85,B 0,C 180,E1 -11191.836,E2 -11191.836} C_VEL
LIN {X 0,Y 397.124,Z 283.641,A -85,B 0,C 180,E1 -11194.493,E2 -11194.493} C_VEL
LIN {X 0,Y 397.102,Z 283.635,A -85,B 0,C 180,E1 -11198.275,E2 -11198.275} C_VEL
LIN {X 0,Y 397.087,Z 283.645,A -85,B 0,C 180,E1 -11200.909,E2 -11200.909} C_VEL
LIN {X 0,Y 397.099,Z 283.646,A -85,B 0,C 180,E1 -11203.649,E2 -11203.649} C_VEL
LIN {X 0,Y 397.1,Z 283.642,A -85,B 0,C 180,E1 -11206.521,E2 -11206.521} C_VEL
LIN {X 0,Y 397.112,Z 283.642,A -85,B 0,C 180,E1 -11210.423,E2 -11210.423} C_VEL
LIN {X 0,Y 397.107,Z 283.647,A -85,B 0,C 180,E1 -11214.266,E2 -11214.266} C_VEL
LIN {X 0,Y 397.179,Z 283.852,A -85,B 0,C 180,E1 -11215.127,E2 -11215.127} C_VEL
LIN {X 0,Y 400.759,Z 297.549,A -85,B 0,C 180,E1 -11218.014,E2 -11218.014} C_VEL
LIN {X 0,Y 403.739,Z 309.968,A -85,B 0,C 180,E1 -11220.501,E2 -11220.501} C_VEL
LIN {X 0,Y 404.295,Z 313.829,A -85,B 0,C 180,E1 -11221.232,E2 -11221.232} C_VEL
LIN {X 0,Y 404.116,Z 315.692,A -85,B 0,C 180,E1 -11221.528,E2 -11221.528} C_VEL
LIN {X 0,Y 408.733,Z 338.434,A -85,B 0,C 180,E1 -11222.317,E2 -11222.317} C_VEL
LIN {X 0,Y 411.392,Z 353.947,A -85,B 0,C 180,E1 -11222.807,E2 -11222.807} C_VEL
LIN {X 0,Y 408.935,Z 477.135,A -85,B 0,C 180,E1 -11224.997,E2 -11224.997} C_VEL
LIN {X 0,Y 408.309,Z 492.592,A -85,B 0,C 180,E1 -11225.398,E2 -11225.398} C_VEL
LIN {X 0,Y 407.332,Z 507.429,A -85,B 0,C 180,E1 -11225.971,E2 -11225.971} C_VEL
LIN {X 0,Y 406.262,Z 521.166,A -85,B 0,C 180,E1 -11226.69,E2 -11226.69} C_VEL
LIN {X 0,Y 404.973,Z 534.272,A -85,B 0,C 180,E1 -11227.556,E2 -11227.556} C_VEL
LIN {X 0,Y 403.526,Z 547.898,A -85,B 0,C 180,E1 -11228.681,E2 -11228.681} C_VEL
LIN {X 0,Y 401.905,Z 561.504,A -85,B 0,C 180,E1 -11230.063,E2 -11230.063} C_VEL
LIN {X 0,Y 400.387,Z 573.75,A -85,B 0,C 180,E1 -11231.582,E2 -11231.582} C_VEL
LIN {X 0,Y 399.228,Z 584.038,A -85,B 0,C 180,E1 -11233.115,E2 -11233.115} C_VEL
LIN {X 0,Y 398.09,Z 594.099,A -85,B 0,C 180,E1 -11234.907,E2 -11234.907} C_VEL
LIN {X 0,Y 397.149,Z 602.571,A -85,B 0,C 180,E1 -11236.726,E2 -11236.726} C_VEL
LIN {X 0,Y 396.558,Z 610.324,A -85,B 0,C 180,E1 -11238.759,E2 -11238.759} C_VEL
LIN {X 0,Y 396.069,Z 616.582,A -85,B 0,C 180,E1 -11240.811,E2 -11240.811} C_VEL
LIN {X 0,Y 395.893,Z 621.43,A -85,B 0,C 180,E1 -11242.862,E2 -11242.862} C_VEL
LIN {X 0,Y 395.769,Z 624.981,A -85,B 0,C 180,E1 -11244.907,E2 -11244.907} C_VEL
LIN {X 0,Y 395.734,Z 627.318,A -85,B 0,C 180,E1 -11246.946,E2 -11246.946} C_VEL
LIN {X 0,Y 395.807,Z 628.497,A -85,B 0,C 180,E1 -11248.983,E2 -11248.983} C_VEL
LIN {X 0,Y 395.808,Z 628.495,A -85,B 0,C 180,E1 -11251.018,E2 -11251.018} C_VEL
LIN {X 0,Y 395.734,Z 627.309,A -85,B 0,C 180,E1 -11253.055,E2 -11253.055} C_VEL
LIN {X 0,Y 395.766,Z 624.967,A -85,B 0,C 180,E1 -11255.094,E2 -11255.094} C_VEL
LIN {X 0,Y 395.892,Z 621.416,A -85,B 0,C 180,E1 -11257.139,E2 -11257.139} C_VEL
LIN {X 0,Y 396.067,Z 616.566,A -85,B 0,C 180,E1 -11259.19,E2 -11259.19} C_VEL
LIN {X 0,Y 396.554,Z 610.294,A -85,B 0,C 180,E1 -11261.242,E2 -11261.242} C_VEL
LIN {X 0,Y 397.153,Z 602.419,A -85,B 0,C 180,E1 -11263.3,E2 -11263.3} C_VEL
LIN {X 0,Y 398.09,Z 594.057,A -85,B 0,C 180,E1 -11265.094,E2 -11265.094} C_VEL
LIN {X 0,Y 399.213,Z 583.986,A -85,B 0,C 180,E1 -11266.887,E2 -11266.887} C_VEL
LIN {X 0,Y 400.492,Z 573.096,A -85,B 0,C 180,E1 -11268.5,E2 -11268.5} C_VEL
LIN {X 0,Y 401.907,Z 561.44,A -85,B 0,C 180,E1 -11269.938,E2 -11269.938} C_VEL
LIN {X 0,Y 403.521,Z 547.806,A -85,B 0,C 180,E1 -11271.32,E2 -11271.32} C_VEL
LIN {X 0,Y 404.963,Z 534.14,A -85,B 0,C 180,E1 -11272.446,E2 -11272.446} C_VEL
LIN {X 0,Y 406.341,Z 519.993,A -85,B 0,C 180,E1 -11273.374,E2 -11273.374} C_VEL
LIN {X 0,Y 407.5,Z 504.541,A -85,B 0,C 180,E1 -11274.154,E2 -11274.154} C_VEL
LIN {X 0,Y 408.448,Z 489.472,A -85,B 0,C 180,E1 -11274.696,E2 -11274.696} C_VEL
LIN {X 0,Y 409.02,Z 473.478,A -85,B 0,C 180,E1 -11275.066,E2 -11275.066} C_VEL
LIN {X 0,Y 411.351,Z 353.389,A -85,B 0,C 180,E1 -11277.197,E2 -11277.197} C_VEL
LIN {X 0,Y 405.67,Z 323.016,A -85,B 0,C 180,E1 -11278.2,E2 -11278.2} C_VEL
LIN {X 0,Y 404.127,Z 315.435,A -85,B 0,C 180,E1 -11278.482,E2 -11278.482} C_VEL
LIN {X 0,Y 404.103,Z 311.75,A -85,B 0,C 180,E1 -11279.142,E2 -11279.142} C_VEL
LIN {X 0,Y 401.659,Z 301.098,A -85,B 0,C 180,E1 -11281.248,E2 -11281.248} C_VEL
LIN {X 0,Y 397.746,Z 285.808,A -85,B 0,C 180,E1 -11284.433,E2 -11284.433} C_VEL
LIN {X 0,Y 397.149,Z 283.641,A -85,B 0,C 180,E1 -11284.954,E2 -11284.954} C_VEL
LIN {X 0,Y 397.127,Z 283.636,A -85,B 0,C 180,E1 -11288.861,E2 -11288.861} C_VEL
LIN {X 0,Y 397.067,Z 283.649,A -85,B 0,C 180,E1 -11292.268,E2 -11292.268} C_VEL
LIN {X 0,Y 397.089,Z 283.645,A -85,B 0,C 180,E1 -11295.069,E2 -11295.069} C_VEL
LIN {X 0,Y 397.069,Z 283.647,A -85,B 0,C 180,E1 -11298.022,E2 -11298.022} C_VEL
LIN {X 0,Y 397.129,Z 283.64,A -85,B 0,C 180,E1 -11301.14,E2 -11301.14} C_VEL
LIN {X 0,Y 397.122,Z 283.639,A -85,B 0,C 180,E1 -11304.497,E2 -11304.497} C_VEL
LIN {X 0,Y 397.082,Z 283.642,A -85,B 0,C 180,E1 -11307.929,E2 -11307.929} C_VEL
LIN {X 0,Y 397.122,Z 283.638,A -85,B 0,C 180,E1 -11310.296,E2 -11310.296} C_VEL
LIN {X 0,Y 397.099,Z 283.64,A -85,B 0,C 180,E1 -11313.739,E2 -11313.739} C_VEL
LIN {X 0,Y 397.108,Z 283.636,A -85,B 0,C 180,E1 -11317.086,E2 -11317.086} C_VEL
LIN {X 0,Y 397.152,Z 283.634,A -85,B 0,C 180,E1 -11320.353,E2 -11320.353} C_VEL
LIN {X 0,Y 397.171,Z 283.636,A -85,B 0,C 180,E1 -11323.553,E2 -11323.553} C_VEL
LIN {X 0,Y 397.234,Z 283.627,A -85,B 0,C 180,E1 -11326.703,E2 -11326.703} C_VEL
LIN {X 0,Y 397.219,Z 283.628,A -85,B 0,C 180,E1 -11329.809,E2 -11329.809} C_VEL
LIN {X 0,Y 397.298,Z 283.611,A -85,B 0,C 180,E1 -11332.887,E2 -11332.887} C_VEL
LIN {X 0,Y 397.237,Z 283.626,A -85,B 0,C 180,E1 -11334.925,E2 -11334.925} C_VEL
LIN {X 0,Y 397.444,Z 283.6,A -85,B 0,C 180,E1 -11337.973,E2 -11337.973} C_VEL
LIN {X 0,Y 397.448,Z 283.598,A -85,B 0,C 180,E1 -11342.027,E2 -11342.027} C_VEL
LIN {X 0,Y 397.297,Z 283.614,A -85,B 0,C 180,E1 -11346.486,E2 -11346.486} C_VEL
LIN {X 0,Y 397.234,Z 283.628,A -85,B 0,C 180,E1 -11349.162,E2 -11349.162} C_VEL
LIN {X 0,Y 397.223,Z 283.629,A -85,B 0,C 180,E1 -11352.258,E2 -11352.258} C_VEL
LIN {X 0,Y 397.127,Z 283.637,A -85,B 0,C 180,E1 -11355.394,E2 -11355.394} C_VEL
LIN {X 0,Y 397.092,Z 283.639,A -85,B 0,C 180,E1 -11358.577,E2 -11358.577} C_VEL
LIN {X 0,Y 397.094,Z 283.643,A -85,B 0,C 180,E1 -11361.819,E2 -11361.819} C_VEL
LIN {X 0,Y 397.105,Z 283.645,A -85,B 0,C 180,E1 -11365.135,E2 -11365.135} C_VEL
LIN {X 0,Y 397.063,Z 283.631,A -85,B 0,C 180,E1 -11368.548,E2 -11368.548} C_VEL
LIN {X 0,Y 397.078,Z 283.647,A -85,B 0,C 180,E1 -11371.834,E2 -11371.834} C_VEL
LIN {X 0,Y 397.118,Z 283.641,A -85,B 0,C 180,E1 -11374.494,E2 -11374.494} C_VEL
LIN {X 0,Y 397.089,Z 283.642,A -85,B 0,C 180,E1 -11378.277,E2 -11378.277} C_VEL
LIN {X 0,Y 397.047,Z 283.651,A -85,B 0,C 180,E1 -11380.914,E2 -11380.914} C_VEL
LIN {X 0,Y 397.041,Z 283.65,A -85,B 0,C 180,E1 -11383.657,E2 -11383.657} C_VEL
LIN {X 0,Y 397.024,Z 283.651,A -85,B 0,C 180,E1 -11386.533,E2 -11386.533} C_VEL
LIN {X 0,Y 397.087,Z 283.644,A -85,B 0,C 180,E1 -11390.419,E2 -11390.419} C_VEL
LIN {X 0,Y 397.093,Z 283.639,A -85,B 0,C 180,E1 -11393.004,E2 -11393.004} C_VEL
LIN {X 0,Y 397.112,Z 283.642,A -85,B 0,C 180,E1 -11396.726,E2 -11396.726} C_VEL
LIN {X 0,Y 397.13,Z 283.789,A -85,B 0,C 180,E1 -11399.815,E2 -11399.815} C_VEL
LIN {X 0,Y 398.657,Z 289.688,A -85,B 0,C 180,E1 -11401.175,E2 -11401.175} C_VEL
LIN {X 0,Y 409.179,Z 312.926,A -85,B 0,C 180,E1 -11402.445,E2 -11402.445} C_VEL
LIN {X 0,Y 411.838,Z 319.12,A -85,B 0,C 180,E1 -11402.76,E2 -11402.76} C_VEL
LIN {X 0,Y 410.043,Z 416.064,A -85,B 0,C 180,E1 -11404.492,E2 -11404.492} C_VEL
LIN {X 0,Y 409.183,Z 453.92,A -85,B 0,C 180,E1 -11405.182,E2 -11405.182} C_VEL
LIN {X 0,Y 408.552,Z 469.135,A -85,B 0,C 180,E1 -11405.646,E2 -11405.646} C_VEL
LIN {X 0,Y 407.711,Z 484.492,A -85,B 0,C 180,E1 -11406.333,E2 -11406.333} C_VEL
LIN {X 0,Y 406.654,Z 497.831,A -85,B 0,C 180,E1 -11407.116,E2 -11407.116} C_VEL
LIN {X 0,Y 405.389,Z 511.397,A -85,B 0,C 180,E1 -11408.115,E2 -11408.115} C_VEL
LIN {X 0,Y 403.851,Z 525.156,A -85,B 0,C 180,E1 -11409.365,E2 -11409.365} C_VEL
LIN {X 0,Y 402.493,Z 537.184,A -85,B 0,C 180,E1 -11410.71,E2 -11410.71} C_VEL
LIN {X 0,Y 401.156,Z 547.936,A -85,B 0,C 180,E1 -11412.146,E2 -11412.146} C_VEL
LIN {X 0,Y 399.965,Z 557.558,A -85,B 0,C 180,E1 -11413.671,E2 -11413.671} C_VEL
LIN {X 0,Y 398.754,Z 566.986,A -85,B 0,C 180,E1 -11415.454,E2 -11415.454} C_VEL
LIN {X 0,Y 397.933,Z 574.834,A -85,B 0,C 180,E1 -11417.248,E2 -11417.248} C_VEL
LIN {X 0,Y 397.046,Z 582.146,A -85,B 0,C 180,E1 -11419.288,E2 -11419.288} C_VEL
LIN {X 0,Y 396.517,Z 587.745,A -85,B 0,C 180,E1 -11421.255,E2 -11421.255} C_VEL
LIN {X 0,Y 395.694,Z 589.731,A -85,B 0,C 180,E1 -11422.051,E2 -11422.051} C_VEL
LIN {X 0,Y 392.627,Z 592.596,A -85,B 0,C 180,E1 -11423.357,E2 -11423.357} C_VEL
LIN {X 0,Y 390.073,Z 594.534,A -85,B 0,C 180,E1 -11424.429,E2 -11424.429} C_VEL
LIN {X 0,Y 388.941,Z 595.751,A -85,B 0,C 180,E1 -11425.268,E2 -11425.268} C_VEL
LIN {X 0,Y 388.826,Z 596.052,A -85,B 0,C 180,E1 -11425.554,E2 -11425.554} C_VEL
LIN {X 0,Y 388.799,Z 597.431,A -85,B 0,C 180,E1 -11426.891,E2 -11426.891} C_VEL
LIN {X 0,Y 388.744,Z 598.606,A -85,B 0,C 180,E1 -11428.964,E2 -11428.964} C_VEL
LIN {X 0,Y 388.745,Z 598.622,A -85,B 0,C 180,E1 -11431.035,E2 -11431.035} C_VEL
LIN {X 0,Y 388.798,Z 597.51,A -85,B 0,C 180,E1 -11433.108,E2 -11433.108} C_VEL
LIN {X 0,Y 388.94,Z 595.271,A -85,B 0,C 180,E1 -11435.183,E2 -11435.183} C_VEL
LIN {X 0,Y 389.14,Z 591.852,A -85,B 0,C 180,E1 -11437.262,E2 -11437.262} C_VEL
LIN {X 0,Y 389.568,Z 587.167,A -85,B 0,C 180,E1 -11439.344,E2 -11439.344} C_VEL
LIN {X 0,Y 390.175,Z 581.093,A -85,B 0,C 180,E1 -11441.428,E2 -11441.428} C_VEL
LIN {X 0,Y 391.045,Z 574.484,A -85,B 0,C 180,E1 -11443.246,E2 -11443.246} C_VEL
LIN {X 0,Y 391.962,Z 566.501,A -85,B 0,C 180,E1 -11445.069,E2 -11445.069} C_VEL
LIN {X 0,Y 393.252,Z 556.911,A -85,B 0,C 180,E1 -11446.882,E2 -11446.882} C_VEL
LIN {X 0,Y 394.522,Z 547.102,A -85,B 0,C 180,E1 -11448.433,E2 -11448.433} C_VEL
LIN {X 0,Y 396.045,Z 535.432,A -85,B 0,C 180,E1 -11449.973,E2 -11449.973} C_VEL
LIN {X 0,Y 397.448,Z 523.804,A -85,B 0,C 180,E1 -11451.253,E2 -11451.253} C_VEL
LIN {X 0,Y 398.866,Z 511.265,A -85,B 0,C 180,E1 -11452.397,E2 -11452.397} C_VEL
LIN {X 0,Y 400.171,Z 497.596,A -85,B 0,C 180,E1 -11453.412,E2 -11453.412} C_VEL
LIN {X 0,Y 401.16,Z 485.42,A -85,B 0,C 180,E1 -11454.139,E2 -11454.139} C_VEL
LIN {X 0,Y 402.137,Z 470.218,A -85,B 0,C 180,E1 -11454.833,E2 -11454.833} C_VEL
LIN {X 0,Y 402.735,Z 455.307,A -85,B 0,C 180,E1 -11455.311,E2 -11455.311} C_VEL
LIN {X 0,Y 403.805,Z 410.867,A -85,B 0,C 180,E1 -11456.139,E2 -11456.139} C_VEL
LIN {X 0,Y 405.554,Z 321.252,A -85,B 0,C 180,E1 -11457.763,E2 -11457.763} C_VEL
LIN {X 0,Y 396.83,Z 301.122,A -85,B 0,C 180,E1 -11458.842,E2 -11458.842} C_VEL
LIN {X 0,Y 391.368,Z 289.596,A -85,B 0,C 180,E1 -11459.559,E2 -11459.559} C_VEL
LIN {X 0,Y 390.039,Z 284.525,A -85,B 0,C 180,E1 -11460.823,E2 -11460.823} C_VEL
LIN {X 0,Y 390.068,Z 284.526,A -85,B 0,C 180,E1 -11464.024,E2 -11464.024} C_VEL
LIN {X 0,Y 390.034,Z 284.528,A -85,B 0,C 180,E1 -11467.78,E2 -11467.78} C_VEL
LIN {X 0,Y 390.014,Z 284.53,A -85,B 0,C 180,E1 -11470.814,E2 -11470.814} C_VEL
LIN {X 0,Y 390.042,Z 284.516,A -85,B 0,C 180,E1 -11473.884,E2 -11473.884} C_VEL
LIN {X 0,Y 390.044,Z 284.514,A -85,B 0,C 180,E1 -11476.788,E2 -11476.788} C_VEL
LIN {X 0,Y 390.007,Z 284.526,A -85,B 0,C 180,E1 -11479.554,E2 -11479.554} C_VEL
LIN {X 0,Y 390.033,Z 284.513,A -85,B 0,C 180,E1 -11482.451,E2 -11482.451} C_VEL
LIN {X 0,Y 390.059,Z 284.518,A -85,B 0,C 180,E1 -11486.044,E2 -11486.044} C_VEL
LIN {X 0,Y 390.038,Z 284.521,A -85,B 0,C 180,E1 -11489.871,E2 -11489.871} C_VEL
LIN {X 0,Y 390.027,Z 284.523,A -85,B 0,C 180,E1 -11493.225,E2 -11493.225} C_VEL
LIN {X 0,Y 390.056,Z 284.517,A -85,B 0,C 180,E1 -11496.767,E2 -11496.767} C_VEL
LIN {X 0,Y 390.068,Z 284.521,A -85,B 0,C 180,E1 -11499.981,E2 -11499.981} C_VEL
LIN {X 0,Y 390.08,Z 284.518,A -85,B 0,C 180,E1 -11503.246,E2 -11503.246} C_VEL
LIN {X 0,Y 390.193,Z 284.501,A -85,B 0,C 180,E1 -11506.561,E2 -11506.561} C_VEL
LIN {X 0,Y 390.16,Z 284.507,A -85,B 0,C 180,E1 -11509.622,E2 -11509.622} C_VEL
LIN {X 0,Y 390.243,Z 284.499,A -85,B 0,C 180,E1 -11512.758,E2 -11512.758} C_VEL
LIN {X 0,Y 390.2,Z 284.498,A -85,B 0,C 180,E1 -11514.833,E2 -11514.833} C_VEL
LIN {X 0,Y 390.412,Z 284.477,A -85,B 0,C 180,E1 -11517.937,E2 -11517.937} C_VEL
LIN {X 0,Y 390.407,Z 284.473,A -85,B 0,C 180,E1 -11522.063,E2 -11522.063} C_VEL
LIN {X 0,Y 390.284,Z 284.488,A -85,B 0,C 180,E1 -11526.202,E2 -11526.202} C_VEL
LIN {X 0,Y 390.191,Z 284.503,A -85,B 0,C 180,E1 -11529.329,E2 -11529.329} C_VEL
LIN {X 0,Y 390.169,Z 284.509,A -85,B 0,C 180,E1 -11532.483,E2 -11532.483} C_VEL
LIN {X 0,Y 390.137,Z 284.506,A -85,B 0,C 180,E1 -11535.677,E2 -11535.677} C_VEL
LIN {X 0,Y 390.103,Z 284.512,A -85,B 0,C 180,E1 -11538.922,E2 -11538.922} C_VEL
LIN {X 0,Y 390.038,Z 284.524,A -85,B 0,C 180,E1 -11542.234,E2 -11542.234} C_VEL
LIN {X 0,Y 390.076,Z 284.496,A -85,B 0,C 180,E1 -11545.62,E2 -11545.62} C_VEL
LIN {X 0,Y 390.032,Z 284.525,A -85,B 0,C 180,E1 -11549.112,E2 -11549.112} C_VEL
LIN {X 0,Y 390.041,Z 284.51,A -85,B 0,C 180,E1 -11552.722,E2 -11552.722} C_VEL
LIN {X 0,Y 390.054,Z 284.519,A -85,B 0,C 180,E1 -11555.825,E2 -11555.825} C_VEL
LIN {X 0,Y 390.069,Z 284.517,A -85,B 0,C 180,E1 -11559.219,E2 -11559.219} C_VEL
LIN {X 0,Y 390.041,Z 284.524,A -85,B 0,C 180,E1 -11562.374,E2 -11562.374} C_VEL
LIN {X 0,Y 390.042,Z 284.523,A -85,B 0,C 180,E1 -11565.355,E2 -11565.355} C_VEL
LIN {X 0,Y 390.029,Z 284.522,A -85,B 0,C 180,E1 -11568.187,E2 -11568.187} C_VEL
LIN {X 0,Y 390.088,Z 284.518,A -85,B 0,C 180,E1 -11570.908,E2 -11570.908} C_VEL
LIN {X 0,Y 390.108,Z 284.605,A -85,B 0,C 180,E1 -11574.604,E2 -11574.604} C_VEL
LIN {X 0,Y 393.515,Z 297.582,A -85,B 0,C 180,E1 -11577.416,E2 -11577.416} C_VEL
LIN {X 0,Y 396.533,Z 309.911,A -85,B 0,C 180,E1 -11579.955,E2 -11579.955} C_VEL
LIN {X 0,Y 397.534,Z 315.206,A -85,B 0,C 180,E1 -11580.999,E2 -11580.999} C_VEL
LIN {X 0,Y 402.602,Z 340.518,A -85,B 0,C 180,E1 -11581.904,E2 -11581.904} C_VEL
LIN {X 0,Y 405.028,Z 354.027,A -85,B 0,C 180,E1 -11582.35,E2 -11582.35} C_VEL
LIN {X 0,Y 402.976,Z 457.641,A -85,B 0,C 180,E1 -11584.221,E2 -11584.221} C_VEL
LIN {X 0,Y 402.328,Z 483.831,A -85,B 0,C 180,E1 -11584.731,E2 -11584.731} C_VEL
LIN {X 0,Y 401.403,Z 499.449,A -85,B 0,C 180,E1 -11585.229,E2 -11585.229} C_VEL
LIN {X 0,Y 400.402,Z 512.784,A -85,B 0,C 180,E1 -11585.828,E2 -11585.828} C_VEL
LIN {X 0,Y 399.122,Z 526.879,A -85,B 0,C 180,E1 -11586.66,E2 -11586.66} C_VEL
LIN {X 0,Y 397.703,Z 540.389,A -85,B 0,C 180,E1 -11587.671,E2 -11587.671} C_VEL
LIN {X 0,Y 396.077,Z 554.15,A -85,B 0,C 180,E1 -11588.942,E2 -11588.942} C_VEL
LIN {X 0,Y 394.501,Z 566.615,A -85,B 0,C 180,E1 -11590.352,E2 -11590.352} C_VEL
LIN {X 0,Y 393.204,Z 577.073,A -85,B 0,C 180,E1 -11591.773,E2 -11591.773} C_VEL
LIN {X 0,Y 391.972,Z 586.786,A -85,B 0,C 180,E1 -11593.329,E2 -11593.329} C_VEL
LIN {X 0,Y 390.868,Z 596.336,A -85,B 0,C 180,E1 -11595.154,E2 -11595.154} C_VEL
LIN {X 0,Y 390.012,Z 604.614,A -85,B 0,C 180,E1 -11597.065,E2 -11597.065} C_VEL
LIN {X 0,Y 389.364,Z 611.737,A -85,B 0,C 180,E1 -11599.075,E2 -11599.075} C_VEL
LIN {X 0,Y 388.928,Z 617.643,A -85,B 0,C 180,E1 -11601.165,E2 -11601.165} C_VEL
LIN {X 0,Y 388.812,Z 621.159,A -85,B 0,C 180,E1 -11602.731,E2 -11602.731} C_VEL
LIN {X 0,Y 388.673,Z 624.71,A -85,B 0,C 180,E1 -11604.813,E2 -11604.813} C_VEL
LIN {X 0,Y 388.639,Z 627.048,A -85,B 0,C 180,E1 -11606.891,E2 -11606.891} C_VEL
LIN {X 0,Y 388.737,Z 628.228,A -85,B 0,C 180,E1 -11608.965,E2 -11608.965} C_VEL
LIN {X 0,Y 388.737,Z 628.226,A -85,B 0,C 180,E1 -11611.036,E2 -11611.036} C_VEL
LIN {X 0,Y 388.639,Z 627.038,A -85,B 0,C 180,E1 -11613.11,E2 -11613.11} C_VEL
LIN {X 0,Y 388.671,Z 624.695,A -85,B 0,C 180,E1 -11615.188,E2 -11615.188} C_VEL
LIN {X 0,Y 388.811,Z 621.144,A -85,B 0,C 180,E1 -11617.27,E2 -11617.27} C_VEL
LIN {X 0,Y 389.004,Z 616.292,A -85,B 0,C 180,E1 -11619.358,E2 -11619.358} C_VEL
LIN {X 0,Y 389.528,Z 610.02,A -85,B 0,C 180,E1 -11621.448,E2 -11621.448} C_VEL
LIN {X 0,Y 390.168,Z 602.143,A -85,B 0,C 180,E1 -11623.543,E2 -11623.543} C_VEL
LIN {X 0,Y 391.163,Z 593.781,A -85,B 0,C 180,E1 -11625.368,E2 -11625.368} C_VEL
LIN {X 0,Y 392.365,Z 583.711,A -85,B 0,C 180,E1 -11627.191,E2 -11627.191} C_VEL
LIN {X 0,Y 393.623,Z 573.419,A -85,B 0,C 180,E1 -11628.747,E2 -11628.747} C_VEL
LIN {X 0,Y 395.197,Z 561.165,A -85,B 0,C 180,E1 -11630.291,E2 -11630.291} C_VEL
LIN {X 0,Y 396.858,Z 547.529,A -85,B 0,C 180,E1 -11631.696,E2 -11631.696} C_VEL
LIN {X 0,Y 398.383,Z 533.864,A -85,B 0,C 180,E1 -11632.837,E2 -11632.837} C_VEL
LIN {X 0,Y 399.852,Z 519.24,A -85,B 0,C 180,E1 -11633.806,E2 -11633.806} C_VEL
LIN {X 0,Y 401.024,Z 504.267,A -85,B 0,C 180,E1 -11634.569,E2 -11634.569} C_VEL
LIN {X 0,Y 401.999,Z 489.188,A -85,B 0,C 180,E1 -11635.12,E2 -11635.12} C_VEL
LIN {X 0,Y 402.608,Z 473.188,A -85,B 0,C 180,E1 -11635.494,E2 -11635.494} C_VEL
LIN {X 0,Y 405.068,Z 355.118,A -85,B 0,C 180,E1 -11637.615,E2 -11637.615} C_VEL
LIN {X 0,Y 400.277,Z 328.744,A -85,B 0,C 180,E1 -11638.495,E2 -11638.495} C_VEL
LIN {X 0,Y 397.512,Z 315.106,A -85,B 0,C 180,E1 -11639.009,E2 -11639.009} C_VEL
LIN {X 0,Y 395.384,Z 304.982,A -85,B 0,C 180,E1 -11641.03,E2 -11641.03} C_VEL
LIN {X 0,Y 391.435,Z 289.39,A -85,B 0,C 180,E1 -11644.32,E2 -11644.32} C_VEL
LIN {X 0,Y 390.093,Z 284.519,A -85,B 0,C 180,E1 -11645.437,E2 -11645.437} C_VEL
LIN {X 0,Y 390.063,Z 284.512,A -85,B 0,C 180,E1 -11649.217,E2 -11649.217} C_VEL
LIN {X 0,Y 390.041,Z 284.525,A -85,B 0,C 180,E1 -11652.374,E2 -11652.374} C_VEL
LIN {X 0,Y 390.047,Z 284.521,A -85,B 0,C 180,E1 -11655.355,E2 -11655.355} C_VEL
LIN {X 0,Y 390.034,Z 284.525,A -85,B 0,C 180,E1 -11658.187,E2 -11658.187} C_VEL
LIN {X 0,Y 390.09,Z 284.517,A -85,B 0,C 180,E1 -11660.908,E2 -11660.908} C_VEL
LIN {X 0,Y 390.088,Z 284.514,A -85,B 0,C 180,E1 -11664.794,E2 -11664.794} C_VEL
LIN {X 0,Y 390.028,Z 284.525,A -85,B 0,C 180,E1 -11668.496,E2 -11668.496} C_VEL
LIN {X 0,Y 390.042,Z 284.523,A -85,B 0,C 180,E1 -11672.064,E2 -11672.064} C_VEL
LIN {X 0,Y 390.064,Z 284.518,A -85,B 0,C 180,E1 -11675.518,E2 -11675.518} C_VEL
LIN {X 0,Y 390.06,Z 284.52,A -85,B 0,C 180,E1 -11678.878,E2 -11678.878} C_VEL
LIN {X 0,Y 390.132,Z 284.514,A -85,B 0,C 180,E1 -11682.167,E2 -11682.167} C_VEL
LIN {X 0,Y 390.149,Z 284.505,A -85,B 0,C 180,E1 -11685.393,E2 -11685.393} C_VEL
LIN {X 0,Y 390.151,Z 284.504,A -85,B 0,C 180,E1 -11688.571,E2 -11688.571} C_VEL
LIN {X 0,Y 390.261,Z 284.493,A -85,B 0,C 180,E1 -11692.086,E2 -11692.086} C_VEL
LIN {X 0,Y 390.209,Z 284.502,A -85,B 0,C 180,E1 -11694.833,E2 -11694.833} C_VEL
LIN {X 0,Y 390.412,Z 284.475,A -85,B 0,C 180,E1 -11697.937,E2 -11697.937} C_VEL
LIN {X 0,Y 390.416,Z 284.474,A -85,B 0,C 180,E1 -11702.063,E2 -11702.063} C_VEL
LIN {X 0,Y 390.258,Z 284.491,A -85,B 0,C 180,E1 -11706.478,E2 -11706.478} C_VEL
LIN {X 0,Y 390.192,Z 284.506,A -85,B 0,C 180,E1 -11709.329,E2 -11709.329} C_VEL
LIN {X 0,Y 390.175,Z 284.506,A -85,B 0,C 180,E1 -11712.483,E2 -11712.483} C_VEL
LIN {X 0,Y 390.068,Z 284.519,A -85,B 0,C 180,E1 -11715.68,E2 -11715.68} C_VEL
LIN {X 0,Y 390.049,Z 284.517,A -85,B 0,C 180,E1 -11718.925,E2 -11718.925} C_VEL
LIN {X 0,Y 390.036,Z 284.519,A -85,B 0,C 180,E1 -11722.235,E2 -11722.235} C_VEL
LIN {X 0,Y 390.054,Z 284.519,A -85,B 0,C 180,E1 -11725.722,E2 -11725.722} C_VEL
LIN {X 0,Y 390.024,Z 284.51,A -85,B 0,C 180,E1 -11729.112,E2 -11729.112} C_VEL
LIN {X 0,Y 390.041,Z 284.521,A -85,B 0,C 180,E1 -11732.722,E2 -11732.722} C_VEL
LIN {X 0,Y 390.044,Z 284.52,A -85,B 0,C 180,E1 -11735.822,E2 -11735.822} C_VEL
LIN {X 0,Y 390.036,Z 284.522,A -85,B 0,C 180,E1 -11739.211,E2 -11739.211} C_VEL
LIN {X 0,Y 390.009,Z 284.525,A -85,B 0,C 180,E1 -11742.368,E2 -11742.368} C_VEL
LIN {X 0,Y 389.993,Z 284.531,A -85,B 0,C 180,E1 -11745.346,E2 -11745.346} C_VEL
LIN {X 0,Y 390.012,Z 284.531,A -85,B 0,C 180,E1 -11749.186,E2 -11749.186} C_VEL
LIN {X 0,Y 390.038,Z 284.519,A -85,B 0,C 180,E1 -11752.451,E2 -11752.451} C_VEL
LIN {X 0,Y 390.064,Z 284.515,A -85,B 0,C 180,E1 -11756.044,E2 -11756.044} C_VEL
LIN {X 0,Y 390.046,Z 284.617,A -85,B 0,C 180,E1 -11759.326,E2 -11759.326} C_VEL
LIN {X 0,Y 391.43,Z 289.854,A -85,B 0,C 180,E1 -11760.588,E2 -11760.588} C_VEL
LIN {X 0,Y 401.919,Z 312.504,A -85,B 0,C 180,E1 -11761.889,E2 -11761.889} C_VEL
LIN {X 0,Y 405.529,Z 321.158,A -85,B 0,C 180,E1 -11762.334,E2 -11762.334} C_VEL
LIN {X 0,Y 403.666,Z 416.359,A -85,B 0,C 180,E1 -11764.059,E2 -11764.059} C_VEL
LIN {X 0,Y 402.742,Z 455.388,A -85,B 0,C 180,E1 -11764.792,E2 -11764.792} C_VEL
LIN {X 0,Y 402.061,Z 470.285,A -85,B 0,C 180,E1 -11765.264,E2 -11765.264} C_VEL
LIN {X 0,Y 401.21,Z 485.108,A -85,B 0,C 180,E1 -11765.945,E2 -11765.945} C_VEL
LIN {X 0,Y 400.136,Z 498.108,A -85,B 0,C 180,E1 -11766.722,E2 -11766.722} C_VEL
LIN {X 0,Y 398.795,Z 511.674,A -85,B 0,C 180,E1 -11767.734,E2 -11767.734} C_VEL
LIN {X 0,Y 397.196,Z 525.432,A -85,B 0,C 180,E1 -11769.003,E2 -11769.003} C_VEL
LIN {X 0,Y 395.726,Z 537.967,A -85,B 0,C 180,E1 -11770.431,E2 -11770.431} C_VEL
LIN {X 0,Y 394.384,Z 548.211,A -85,B 0,C 180,E1 -11771.828,E2 -11771.828} C_VEL
LIN {X 0,Y 393.128,Z 557.833,A -85,B 0,C 180,E1 -11773.379,E2 -11773.379} C_VEL
LIN {X 0,Y 391.852,Z 567.26,A -85,B 0,C 180,E1 -11775.192,E2 -11775.192} C_VEL
LIN {X 0,Y 390.969,Z 575.099,A -85,B 0,C 180,E1 -11777.014,E2 -11777.014} C_VEL
LIN {X 0,Y 390.056,Z 582.418,A -85,B 0,C 180,E1 -11779.094,E2 -11779.094} C_VEL
LIN {X 0,Y 389.471,Z 588.246,A -85,B 0,C 180,E1 -11781.188,E2 -11781.188} C_VEL
LIN {X 0,Y 389.105,Z 592.935,A -85,B 0,C 180,E1 -11783.418,E2 -11783.418} C_VEL
LIN {X 0,Y 388.826,Z 596.052,A -85,B 0,C 180,E1 -11785.554,E2 -11785.554} C_VEL
LIN {X 0,Y 388.092,Z 597.055,A -85,B 0,C 180,E1 -11786.406,E2 -11786.406} C_VEL
LIN {X 0,Y 385.196,Z 598.329,A -85,B 0,C 180,E1 -11787.799,E2 -11787.799} C_VEL
LIN {X 0,Y 382.78,Z 598.909,A -85,B 0,C 180,E1 -11788.931,E2 -11788.931} C_VEL
LIN {X 0,Y 381.74,Z 599.041,A -85,B 0,C 180,E1 -11789.808,E2 -11789.808} C_VEL
LIN {X 0,Y 381.652,Z 599.018,A -85,B 0,C 180,E1 -11790.105,E2 -11790.105} C_VEL
LIN {X 0,Y 381.727,Z 598.472,A -85,B 0,C 180,E1 -11792.11,E2 -11792.11} C_VEL
LIN {X 0,Y 381.724,Z 596.806,A -85,B 0,C 180,E1 -11794.223,E2 -11794.223} C_VEL
LIN {X 0,Y 381.976,Z 593.983,A -85,B 0,C 180,E1 -11796.338,E2 -11796.338} C_VEL
LIN {X 0,Y 382.285,Z 589.944,A -85,B 0,C 180,E1 -11798.457,E2 -11798.457} C_VEL
LIN {X 0,Y 382.852,Z 584.583,A -85,B 0,C 180,E1 -11800.577,E2 -11800.577} C_VEL
LIN {X 0,Y 383.746,Z 577.744,A -85,B 0,C 180,E1 -11802.695,E2 -11802.695} C_VEL
LIN {X 0,Y 384.606,Z 570.361,A -85,B 0,C 180,E1 -11804.559,E2 -11804.559} C_VEL
LIN {X 0,Y 385.863,Z 561.523,A -85,B 0,C 180,E1 -11806.398,E2 -11806.398} C_VEL
LIN {X 0,Y 387.109,Z 552.476,A -85,B 0,C 180,E1 -11807.977,E2 -11807.977} C_VEL
LIN {X 0,Y 388.645,Z 541.314,A -85,B 0,C 180,E1 -11809.613,E2 -11809.613} C_VEL
LIN {X 0,Y 390.15,Z 528.972,A -85,B 0,C 180,E1 -11811.116,E2 -11811.116} C_VEL
LIN {X 0,Y 391.84,Z 515.972,A -85,B 0,C 180,E1 -11812.404,E2 -11812.404} C_VEL
LIN {X 0,Y 393.147,Z 503.321,A -85,B 0,C 180,E1 -11813.437,E2 -11813.437} C_VEL
LIN {X 0,Y 394.432,Z 489.865,A -85,B 0,C 180,E1 -11814.317,E2 -11814.317} C_VEL
LIN {X 0,Y 395.364,Z 475.352,A -85,B 0,C 180,E1 -11815.063,E2 -11815.063} C_VEL
LIN {X 0,Y 396.166,Z 460.111,A -85,B 0,C 180,E1 -11815.62,E2 -11815.62} C_VEL
LIN {X 0,Y 396.657,Z 445.056,A -85,B 0,C 180,E1 -11815.974,E2 -11815.974} C_VEL
LIN {X 0,Y 398.942,Z 342.486,A -85,B 0,C 180,E1 -11817.844,E2 -11817.844} C_VEL
LIN {X 0,Y 399.25,Z 323.057,A -85,B 0,C 180,E1 -11818.209,E2 -11818.209} C_VEL
LIN {X 0,Y 390.645,Z 303.379,A -85,B 0,C 180,E1 -11819.301,E2 -11819.301} C_VEL
LIN {X 0,Y 384.184,Z 289.98,A -85,B 0,C 180,E1 -11820.15,E2 -11820.15} C_VEL
LIN {X 0,Y 382.97,Z 285.408,A -85,B 0,C 180,E1 -11821.303,E2 -11821.303} C_VEL
LIN {X 0,Y 383.009,Z 285.409,A -85,B 0,C 180,E1 -11824.668,E2 -11824.668} C_VEL
LIN {X 0,Y 382.99,Z 285.405,A -85,B 0,C 180,E1 -11827.902,E2 -11827.902} C_VEL
LIN {X 0,Y 382.958,Z 285.407,A -85,B 0,C 180,E1 -11831.35,E2 -11831.35} C_VEL
LIN {X 0,Y 382.987,Z 285.397,A -85,B 0,C 180,E1 -11834.302,E2 -11834.302} C_VEL
LIN {X 0,Y 382.979,Z 285.389,A -85,B 0,C 180,E1 -11837.236,E2 -11837.236} C_VEL
LIN {X 0,Y 382.981,Z 285.404,A -85,B 0,C 180,E1 -11840.419,E2 -11840.419} C_VEL
LIN {X 0,Y 383.009,Z 285.376,A -85,B 0,C 180,E1 -11844.043,E2 -11844.043} C_VEL
LIN {X 0,Y 382.979,Z 285.402,A -85,B 0,C 180,E1 -11847.579,E2 -11847.579} C_VEL
LIN {X 0,Y 382.971,Z 285.405,A -85,B 0,C 180,E1 -11850.298,E2 -11850.298} C_VEL
LIN {X 0,Y 383,Z 285.399,A -85,B 0,C 180,E1 -11854.045,E2 -11854.045} C_VEL
LIN {X 0,Y 382.982,Z 285.398,A -85,B 0,C 180,E1 -11857.333,E2 -11857.333} C_VEL
LIN {X 0,Y 383.011,Z 285.393,A -85,B 0,C 180,E1 -11860.714,E2 -11860.714} C_VEL
LIN {X 0,Y 383.009,Z 285.401,A -85,B 0,C 180,E1 -11864.023,E2 -11864.023} C_VEL
LIN {X 0,Y 383.134,Z 285.381,A -85,B 0,C 180,E1 -11867.284,E2 -11867.284} C_VEL
LIN {X 0,Y 383.137,Z 285.376,A -85,B 0,C 180,E1 -11870.497,E2 -11870.497} C_VEL
LIN {X 0,Y 383.23,Z 285.372,A -85,B 0,C 180,E1 -11873.683,E2 -11873.683} C_VEL
LIN {X 0,Y 383.378,Z 285.353,A -85,B 0,C 180,E1 -11877.899,E2 -11877.899} C_VEL
LIN {X 0,Y 383.373,Z 285.349,A -85,B 0,C 180,E1 -11882.101,E2 -11882.101} C_VEL
LIN {X 0,Y 383.24,Z 285.365,A -85,B 0,C 180,E1 -11886.317,E2 -11886.317} C_VEL
LIN {X 0,Y 383.141,Z 285.382,A -85,B 0,C 180,E1 -11889.502,E2 -11889.502} C_VEL
LIN {X 0,Y 383.124,Z 285.387,A -85,B 0,C 180,E1 -11893.536,E2 -11893.536} C_VEL
LIN {X 0,Y 383.093,Z 285.39,A -85,B 0,C 180,E1 -11897.454,E2 -11897.454} C_VEL
LIN {X 0,Y 383.027,Z 285.397,A -85,B 0,C 180,E1 -11900.647,E2 -11900.647} C_VEL
LIN {X 0,Y 383.026,Z 285.383,A -85,B 0,C 180,E1 -11903.808,E2 -11903.808} C_VEL
LIN {X 0,Y 382.992,Z 285.395,A -85,B 0,C 180,E1 -11907.307,E2 -11907.307} C_VEL
LIN {X 0,Y 382.98,Z 285.392,A -85,B 0,C 180,E1 -11910.919,E2 -11910.919} C_VEL
LIN {X 0,Y 383.016,Z 285.398,A -85,B 0,C 180,E1 -11914.668,E2 -11914.668} C_VEL
LIN {X 0,Y 382.998,Z 285.388,A -85,B 0,C 180,E1 -11917.904,E2 -11917.904} C_VEL
LIN {X 0,Y 382.982,Z 285.403,A -85,B 0,C 180,E1 -11921.347,E2 -11921.347} C_VEL
LIN {X 0,Y 382.994,Z 285.401,A -85,B 0,C 180,E1 -11924.304,E2 -11924.304} C_VEL
LIN {X 0,Y 383.008,Z 285.398,A -85,B 0,C 180,E1 -11927.24,E2 -11927.24} C_VEL
LIN {X 0,Y 383.013,Z 285.399,A -85,B 0,C 180,E1 -11930.414,E2 -11930.414} C_VEL
LIN {X 0,Y 383.041,Z 285.591,A -85,B 0,C 180,E1 -11934.108,E2 -11934.108} C_VEL
LIN {X 0,Y 386.319,Z 297.677,A -85,B 0,C 180,E1 -11936.808,E2 -11936.808} C_VEL
LIN {X 0,Y 389.891,Z 312.392,A -85,B 0,C 180,E1 -11939.908,E2 -11939.908} C_VEL
LIN {X 0,Y 390.444,Z 314.9,A -85,B 0,C 180,E1 -11940.42,E2 -11940.42} C_VEL
LIN {X 0,Y 391.874,Z 319.391,A -85,B 0,C 180,E1 -11940.639,E2 -11940.639} C_VEL
LIN {X 0,Y 396.428,Z 342.21,A -85,B 0,C 180,E1 -11941.466,E2 -11941.466} C_VEL
LIN {X 0,Y 398.755,Z 356.236,A -85,B 0,C 180,E1 -11941.926,E2 -11941.926} C_VEL
LIN {X 0,Y 396.267,Z 471.717,A -85,B 0,C 180,E1 -11944.034,E2 -11944.034} C_VEL
LIN {X 0,Y 395.676,Z 488.137,A -85,B 0,C 180,E1 -11944.416,E2 -11944.416} C_VEL
LIN {X 0,Y 394.673,Z 503.386,A -85,B 0,C 180,E1 -11944.971,E2 -11944.971} C_VEL
LIN {X 0,Y 393.473,Z 517.487,A -85,B 0,C 180,E1 -11945.682,E2 -11945.682} C_VEL
LIN {X 0,Y 392.184,Z 530.303,A -85,B 0,C 180,E1 -11946.511,E2 -11946.511} C_VEL
LIN {X 0,Y 390.55,Z 544.498,A -85,B 0,C 180,E1 -11947.658,E2 -11947.658} C_VEL
LIN {X 0,Y 388.951,Z 557.458,A -85,B 0,C 180,E1 -11948.954,E2 -11948.954} C_VEL
LIN {X 0,Y 387.42,Z 569.336,A -85,B 0,C 180,E1 -11950.392,E2 -11950.392} C_VEL
LIN {X 0,Y 386.172,Z 578.643,A -85,B 0,C 180,E1 -11951.715,E2 -11951.715} C_VEL
LIN {X 0,Y 384.785,Z 589.46,A -85,B 0,C 180,E1 -11953.555,E2 -11953.555} C_VEL
LIN {X 0,Y 383.615,Z 598.53,A -85,B 0,C 180,E1 -11955.41,E2 -11955.41} C_VEL
LIN {X 0,Y 382.848,Z 606.064,A -85,B 0,C 180,E1 -11957.275,E2 -11957.275} C_VEL
LIN {X 0,Y 382.147,Z 613.094,A -85,B 0,C 180,E1 -11959.403,E2 -11959.403} C_VEL
LIN {X 0,Y 381.797,Z 618.63,A -85,B 0,C 180,E1 -11961.532,E2 -11961.532} C_VEL
LIN {X 0,Y 381.653,Z 623.283,A -85,B 0,C 180,E1 -11963.927,E2 -11963.927} C_VEL
LIN {X 0,Y 381.594,Z 625.758,A -85,B 0,C 180,E1 -11965.776,E2 -11965.776} C_VEL
LIN {X 0,Y 381.601,Z 627.511,A -85,B 0,C 180,E1 -11967.89,E2 -11967.89} C_VEL
LIN {X 0,Y 381.654,Z 628.113,A -85,B 0,C 180,E1 -11970.001,E2 -11970.001} C_VEL
LIN {X 0,Y 381.601,Z 627.505,A -85,B 0,C 180,E1 -11972.111,E2 -11972.111} C_VEL
LIN {X 0,Y 381.593,Z 625.744,A -85,B 0,C 180,E1 -11974.225,E2 -11974.225} C_VEL
LIN {X 0,Y 381.66,Z 622.803,A -85,B 0,C 180,E1 -11976.344,E2 -11976.344} C_VEL
LIN {X 0,Y 381.796,Z 618.613,A -85,B 0,C 180,E1 -11978.469,E2 -11978.469} C_VEL
LIN {X 0,Y 382.143,Z 613.068,A -85,B 0,C 180,E1 -11980.598,E2 -11980.598} C_VEL
LIN {X 0,Y 382.849,Z 606.022,A -85,B 0,C 180,E1 -11982.726,E2 -11982.726} C_VEL
LIN {X 0,Y 383.617,Z 598.485,A -85,B 0,C 180,E1 -11984.591,E2 -11984.591} C_VEL
LIN {X 0,Y 384.72,Z 589.409,A -85,B 0,C 180,E1 -11986.449,E2 -11986.449} C_VEL
LIN {X 0,Y 386.213,Z 578.561,A -85,B 0,C 180,E1 -11988.287,E2 -11988.287} C_VEL
LIN {X 0,Y 387.613,Z 567.491,A -85,B 0,C 180,E1 -11989.848,E2 -11989.848} C_VEL
LIN {X 0,Y 389.249,Z 555.015,A -85,B 0,C 180,E1 -11991.307,E2 -11991.307} C_VEL
LIN {X 0,Y 390.925,Z 541.52,A -85,B 0,C 180,E1 -11992.599,E2 -11992.599} C_VEL
LIN {X 0,Y 392.358,Z 528.462,A -85,B 0,C 180,E1 -11993.613,E2 -11993.613} C_VEL
LIN {X 0,Y 393.763,Z 514.243,A -85,B 0,C 180,E1 -11994.49,E2 -11994.49} C_VEL
LIN {X 0,Y 394.872,Z 499.787,A -85,B 0,C 180,E1 -11995.172,E2 -11995.172} C_VEL
LIN {X 0,Y 395.822,Z 484.334,A -85,B 0,C 180,E1 -11995.681,E2 -11995.681} C_VEL
LIN {X 0,Y 396.49,Z 460.358,A -85,B 0,C 180,E1 -11996.163,E2 -11996.163} C_VEL
LIN {X 0,Y 398.636,Z 354.969,A -85,B 0,C 180,E1 -11998.097,E2 -11998.097} C_VEL
LIN {X 0,Y 393.322,Z 326.362,A -85,B 0,C 180,E1 -11999.088,E2 -11999.088} C_VEL
LIN {X 0,Y 391.191,Z 317.028,A -85,B 0,C 180,E1 -11999.452,E2 -11999.452} C_VEL
LIN {X 0,Y 390.398,Z 314.887,A -85,B 0,C 180,E1 -11999.573,E2 -11999.573} C_VEL
LIN {X 0,Y 388.044,Z 304.666,A -85,B 0,C 180,E1 -12001.684,E2 -12001.684} C_VEL
LIN {X 0,Y 384.558,Z 290.856,A -85,B 0,C 180,E1 -12004.675,E2 -12004.675} C_VEL
LIN {X 0,Y 383.027,Z 285.4,A -85,B 0,C 180,E1 -12005.956,E2 -12005.956} C_VEL
LIN {X 0,Y 383.012,Z 285.39,A -85,B 0,C 180,E1 -12009.586,E2 -12009.586} C_VEL
LIN {X 0,Y 383.008,Z 285.402,A -85,B 0,C 180,E1 -12012.779,E2 -12012.779} C_VEL
LIN {X 0,Y 382.999,Z 285.395,A -85,B 0,C 180,E1 -12015.79,E2 -12015.79} C_VEL
LIN {X 0,Y 382.991,Z 285.402,A -85,B 0,C 180,E1 -12018.796,E2 -12018.796} C_VEL
LIN {X 0,Y 383.001,Z 285.399,A -85,B 0,C 180,E1 -12022.097,E2 -12022.097} C_VEL
LIN {X 0,Y 383.021,Z 285.393,A -85,B 0,C 180,E1 -12025.333,E2 -12025.333} C_VEL
LIN {X 0,Y 382.986,Z 285.399,A -85,B 0,C 180,E1 -12029.082,E2 -12029.082} C_VEL
LIN {X 0,Y 382.997,Z 285.397,A -85,B 0,C 180,E1 -12032.694,E2 -12032.694} C_VEL
LIN {X 0,Y 383.021,Z 285.397,A -85,B 0,C 180,E1 -12036.192,E2 -12036.192} C_VEL
LIN {X 0,Y 383.06,Z 285.393,A -85,B 0,C 180,E1 -12039.599,E2 -12039.599} C_VEL
LIN {X 0,Y 383.11,Z 285.386,A -85,B 0,C 180,E1 -12042.932,E2 -12042.932} C_VEL
LIN {X 0,Y 383.13,Z 285.385,A -85,B 0,C 180,E1 -12046.464,E2 -12046.464} C_VEL
LIN {X 0,Y 383.147,Z 285.383,A -85,B 0,C 180,E1 -12050.498,E2 -12050.498} C_VEL
LIN {X 0,Y 383.244,Z 285.365,A -85,B 0,C 180,E1 -12053.683,E2 -12053.683} C_VEL
LIN {X 0,Y 383.378,Z 285.351,A -85,B 0,C 180,E1 -12057.899,E2 -12057.899} C_VEL
LIN {X 0,Y 383.382,Z 285.35,A -85,B 0,C 180,E1 -12062.101,E2 -12062.101} C_VEL
LIN {X 0,Y 383.223,Z 285.368,A -85,B 0,C 180,E1 -12066.466,E2 -12066.466} C_VEL
LIN {X 0,Y 383.143,Z 285.383,A -85,B 0,C 180,E1 -12069.502,E2 -12069.502} C_VEL
LIN {X 0,Y 383.131,Z 285.386,A -85,B 0,C 180,E1 -12073.536,E2 -12073.536} C_VEL
LIN {X 0,Y 383.028,Z 285.401,A -85,B 0,C 180,E1 -12077.42,E2 -12077.42} C_VEL
LIN {X 0,Y 383.018,Z 285.398,A -85,B 0,C 180,E1 -12080.64,E2 -12080.64} C_VEL
LIN {X 0,Y 383.011,Z 285.402,A -85,B 0,C 180,E1 -12083.809,E2 -12083.809} C_VEL
LIN {X 0,Y 382.969,Z 285.388,A -85,B 0,C 180,E1 -12087.309,E2 -12087.309} C_VEL
LIN {X 0,Y 382.981,Z 285.402,A -85,B 0,C 180,E1 -12090.919,E2 -12090.919} C_VEL
LIN {X 0,Y 383.014,Z 285.398,A -85,B 0,C 180,E1 -12094.669,E2 -12094.669} C_VEL
LIN {X 0,Y 382.993,Z 285.399,A -85,B 0,C 180,E1 -12097.901,E2 -12097.901} C_VEL
LIN {X 0,Y 382.958,Z 285.404,A -85,B 0,C 180,E1 -12101.351,E2 -12101.351} C_VEL
LIN {X 0,Y 382.966,Z 285.402,A -85,B 0,C 180,E1 -12104.298,E2 -12104.298} C_VEL
LIN {X 0,Y 382.949,Z 285.41,A -85,B 0,C 180,E1 -12107.231,E2 -12107.231} C_VEL
LIN {X 0,Y 382.985,Z 285.401,A -85,B 0,C 180,E1 -12110.419,E2 -12110.419} C_VEL
LIN {X 0,Y 383.014,Z 285.401,A -85,B 0,C 180,E1 -12114.043,E2 -12114.043} C_VEL
LIN {X 0,Y 382.983,Z 285.403,A -85,B 0,C 180,E1 -12117.579,E2 -12117.579} C_VEL
LIN {X 0,Y 383.002,Z 285.576,A -85,B 0,C 180,E1 -12118.852,E2 -12118.852} C_VEL
LIN {X 0,Y 384.259,Z 290.187,A -85,B 0,C 180,E1 -12119.983,E2 -12119.983} C_VEL
LIN {X 0,Y 393.575,Z 309.795,A -85,B 0,C 180,E1 -12121.174,E2 -12121.174} C_VEL
LIN {X 0,Y 399.225,Z 322.942,A -85,B 0,C 180,E1 -12121.889,E2 -12121.889} C_VEL
LIN {X 0,Y 397.308,Z 416.654,A -85,B 0,C 180,E1 -12123.612,E2 -12123.612} C_VEL
LIN {X 0,Y 396.358,Z 454.498,A -85,B 0,C 180,E1 -12124.321,E2 -12124.321} C_VEL
LIN {X 0,Y 395.691,Z 469.818,A -85,B 0,C 180,E1 -12124.806,E2 -12124.806} C_VEL
LIN {X 0,Y 394.806,Z 484.691,A -85,B 0,C 180,E1 -12125.489,E2 -12125.489} C_VEL
LIN {X 0,Y 393.631,Z 498.385,A -85,B 0,C 180,E1 -12126.314,E2 -12126.314} C_VEL
LIN {X 0,Y 392.24,Z 511.95,A -85,B 0,C 180,E1 -12127.341,E2 -12127.341} C_VEL
LIN {X 0,Y 390.56,Z 525.708,A -85,B 0,C 180,E1 -12128.629,E2 -12128.629} C_VEL
LIN {X 0,Y 389.131,Z 537.047,A -85,B 0,C 180,E1 -12129.93,E2 -12129.93} C_VEL
LIN {X 0,Y 387.624,Z 548.485,A -85,B 0,C 180,E1 -12131.5,E2 -12131.5} C_VEL
LIN {X 0,Y 386.298,Z 558.107,A -85,B 0,C 180,E1 -12133.076,E2 -12133.076} C_VEL
LIN {X 0,Y 384.962,Z 567.534,A -85,B 0,C 180,E1 -12134.92,E2 -12134.92} C_VEL
LIN {X 0,Y 384.022,Z 575.372,A -85,B 0,C 180,E1 -12136.775,E2 -12136.775} C_VEL
LIN {X 0,Y 383.043,Z 582.692,A -85,B 0,C 180,E1 -12138.892,E2 -12138.892} C_VEL
LIN {X 0,Y 382.43,Z 588.493,A -85,B 0,C 180,E1 -12141.013,E2 -12141.013} C_VEL
LIN {X 0,Y 382.113,Z 591.926,A -85,B 0,C 180,E1 -12142.602,E2 -12142.602} C_VEL
LIN {X 0,Y 381.888,Z 595.401,A -85,B 0,C 180,E1 -12144.72,E2 -12144.72} C_VEL
LIN {X 0,Y 381.703,Z 597.702,A -85,B 0,C 180,E1 -12146.833,E2 -12146.833} C_VEL
LIN {X 0,Y 381.677,Z 598.875,A -85,B 0,C 180,E1 -12148.944,E2 -12148.944} C_VEL
LIN {X 0,Y 381.652,Z 599.018,A -85,B 0,C 180,E1 -12150.105,E2 -12150.105} C_VEL
LIN {X 0,Y 380.965,Z 598.935,A -85,B 0,C 180,E1 -12150.987,E2 -12150.987} C_VEL
LIN {X 0,Y 378.09,Z 598.48,A -85,B 0,C 180,E1 -12152.419,E2 -12152.419} C_VEL
LIN {X 0,Y 375.709,Z 597.749,A -85,B 0,C 180,E1 -12153.572,E2 -12153.572} C_VEL
LIN {X 0,Y 374.749,Z 596.911,A -85,B 0,C 180,E1 -12154.459,E2 -12154.459} C_VEL
LIN {X 0,Y 374.703,Z 596.542,A -85,B 0,C 180,E1 -12154.757,E2 -12154.757} C_VEL
LIN {X 0,Y 374.944,Z 594.074,A -85,B 0,C 180,E1 -12156.566,E2 -12156.566} C_VEL
LIN {X 0,Y 375.255,Z 590.214,A -85,B 0,C 180,E1 -12158.617,E2 -12158.617} C_VEL
LIN {X 0,Y 375.858,Z 584.853,A -85,B 0,C 180,E1 -12160.776,E2 -12160.776} C_VEL
LIN {X 0,Y 376.778,Z 578.014,A -85,B 0,C 180,E1 -12162.934,E2 -12162.934} C_VEL
LIN {X 0,Y 377.566,Z 571.393,A -85,B 0,C 180,E1 -12164.647,E2 -12164.647} C_VEL
LIN {X 0,Y 378.815,Z 563.134,A -85,B 0,C 180,E1 -12166.434,E2 -12166.434} C_VEL
LIN {X 0,Y 380.321,Z 552.745,A -85,B 0,C 180,E1 -12168.309,E2 -12168.309} C_VEL
LIN {X 0,Y 381.887,Z 541.961,A -85,B 0,C 180,E1 -12169.92,E2 -12169.92} C_VEL
LIN {X 0,Y 383.368,Z 530.405,A -85,B 0,C 180,E1 -12171.367,E2 -12171.367} C_VEL
LIN {X 0,Y 385.117,Z 517.656,A -85,B 0,C 180,E1 -12172.675,E2 -12172.675} C_VEL
LIN {X 0,Y 386.48,Z 505.343,A -85,B 0,C 180,E1 -12173.724,E2 -12173.724} C_VEL
LIN {X 0,Y 387.712,Z 492.126,A -85,B 0,C 180,E1 -12174.64,E2 -12174.64} C_VEL
LIN {X 0,Y 388.894,Z 476.956,A -85,B 0,C 180,E1 -12175.446,E2 -12175.446} C_VEL
LIN {X 0,Y 389.743,Z 461.502,A -85,B 0,C 180,E1 -12176.038,E2 -12176.038} C_VEL
LIN {X 0,Y 390.261,Z 447.086,A -85,B 0,C 180,E1 -12176.396,E2 -12176.396} C_VEL
LIN {X 0,Y 392.707,Z 342.079,A -85,B 0,C 180,E1 -12178.339,E2 -12178.339} C_VEL
LIN {X 0,Y 393.014,Z 325.024,A -85,B 0,C 180,E1 -12178.662,E2 -12178.662} C_VEL
LIN {X 0,Y 384.8,Z 306.335,A -85,B 0,C 180,E1 -12179.734,E2 -12179.734} C_VEL
LIN {X 0,Y 376.972,Z 290.232,A -85,B 0,C 180,E1 -12180.801,E2 -12180.801} C_VEL
LIN {X 0,Y 375.972,Z 286.285,A -85,B 0,C 180,E1 -12181.836,E2 -12181.836} C_VEL
LIN {X 0,Y 375.947,Z 286.279,A -85,B 0,C 180,E1 -12185.416,E2 -12185.416} C_VEL
LIN {X 0,Y 375.933,Z 286.284,A -85,B 0,C 180,E1 -12188.262,E2 -12188.262} C_VEL
LIN {X 0,Y 375.911,Z 286.283,A -85,B 0,C 180,E1 -12191.597,E2 -12191.597} C_VEL
LIN {X 0,Y 375.918,Z 286.282,A -85,B 0,C 180,E1 -12194.73,E2 -12194.73} C_VEL
LIN {X 0,Y 375.905,Z 286.267,A -85,B 0,C 180,E1 -12197.696,E2 -12197.696} C_VEL
LIN {X 0,Y 375.93,Z 286.284,A -85,B 0,C 180,E1 -12200.533,E2 -12200.533} C_VEL
LIN {X 0,Y 375.954,Z 286.254,A -85,B 0,C 180,E1 -12203.497,E2 -12203.497} C_VEL
LIN {X 0,Y 375.955,Z 286.274,A -85,B 0,C 180,E1 -12205.888,E2 -12205.888} C_VEL
LIN {X 0,Y 375.957,Z 286.275,A -85,B 0,C 180,E1 -12209.687,E2 -12209.687} C_VEL
LIN {X 0,Y 375.915,Z 286.281,A -85,B 0,C 180,E1 -12212.135,E2 -12212.135} C_VEL
LIN {X 0,Y 375.934,Z 286.285,A -85,B 0,C 180,E1 -12214.534,E2 -12214.534} C_VEL
LIN {X 0,Y 375.967,Z 286.272,A -85,B 0,C 180,E1 -12216.886,E2 -12216.886} C_VEL
LIN {X 0,Y 375.958,Z 286.275,A -85,B 0,C 180,E1 -12220.337,E2 -12220.337} C_VEL
LIN {X 0,Y 375.958,Z 286.278,A -85,B 0,C 180,E1 -12223.716,E2 -12223.716} C_VEL
LIN {X 0,Y 376.102,Z 286.258,A -85,B 0,C 180,E1 -12227.042,E2 -12227.042} C_VEL
LIN {X 0,Y 376.108,Z 286.253,A -85,B 0,C 180,E1 -12230.318,E2 -12230.318} C_VEL
LIN {X 0,Y 376.19,Z 286.249,A -85,B 0,C 180,E1 -12233.564,E2 -12233.564} C_VEL
LIN {X 0,Y 376.342,Z 286.229,A -85,B 0,C 180,E1 -12237.859,E2 -12237.859} C_VEL
LIN {X 0,Y 376.338,Z 286.226,A -85,B 0,C 180,E1 -12242.14,E2 -12242.14} C_VEL
LIN {X 0,Y 376.198,Z 286.242,A -85,B 0,C 180,E1 -12246.436,E2 -12246.436} C_VEL
LIN {X 0,Y 376.111,Z 286.259,A -85,B 0,C 180,E1 -12249.682,E2 -12249.682} C_VEL
LIN {X 0,Y 376.088,Z 286.264,A -85,B 0,C 180,E1 -12253.658,E2 -12253.658} C_VEL
LIN {X 0,Y 376.041,Z 286.27,A -85,B 0,C 180,E1 -12257.607,E2 -12257.607} C_VEL
LIN {X 0,Y 375.976,Z 286.275,A -85,B 0,C 180,E1 -12260.832,E2 -12260.832} C_VEL
LIN {X 0,Y 375.981,Z 286.254,A -85,B 0,C 180,E1 -12264.282,E2 -12264.282} C_VEL
LIN {X 0,Y 375.933,Z 286.28,A -85,B 0,C 180,E1 -12267.864,E2 -12267.864} C_VEL
LIN {X 0,Y 375.955,Z 286.26,A -85,B 0,C 180,E1 -12271.562,E2 -12271.562} C_VEL
LIN {X 0,Y 375.956,Z 286.281,A -85,B 0,C 180,E1 -12275.416,E2 -12275.416} C_VEL
LIN {X 0,Y 375.973,Z 286.265,A -85,B 0,C 180,E1 -12278.271,E2 -12278.271} C_VEL
LIN {X 0,Y 375.933,Z 286.282,A -85,B 0,C 180,E1 -12281.601,E2 -12281.601} C_VEL
LIN {X 0,Y 375.925,Z 286.281,A -85,B 0,C 180,E1 -12285.269,E2 -12285.269} C_VEL
LIN {X 0,Y 375.932,Z 286.277,A -85,B 0,C 180,E1 -12288.399,E2 -12288.399} C_VEL
LIN {X 0,Y 375.972,Z 286.277,A -85,B 0,C 180,E1 -12291.73,E2 -12291.73} C_VEL
LIN {X 0,Y 375.978,Z 286.362,A -85,B 0,C 180,E1 -12293.546,E2 -12293.546} C_VEL
LIN {X 0,Y 379.443,Z 299.055,A -85,B 0,C 180,E1 -12296.458,E2 -12296.458} C_VEL
LIN {X 0,Y 383.086,Z 314.122,A -85,B 0,C 180,E1 -12299.704,E2 -12299.704} C_VEL
LIN {X 0,Y 383.35,Z 315.05,A -85,B 0,C 180,E1 -12299.835,E2 -12299.835} C_VEL
LIN {X 0,Y 385.869,Z 321.601,A -85,B 0,C 180,E1 -12300.187,E2 -12300.187} C_VEL
LIN {X 0,Y 390.259,Z 343.684,A -85,B 0,C 180,E1 -12301.008,E2 -12301.008} C_VEL
LIN {X 0,Y 392.477,Z 357.211,A -85,B 0,C 180,E1 -12301.461,E2 -12301.461} C_VEL
LIN {X 0,Y 389.889,Z 471.467,A -85,B 0,C 180,E1 -12303.577,E2 -12303.577} C_VEL
LIN {X 0,Y 389.283,Z 487.879,A -85,B 0,C 180,E1 -12303.965,E2 -12303.965} C_VEL
LIN {X 0,Y 388.209,Z 503.358,A -85,B 0,C 180,E1 -12304.536,E2 -12304.536} C_VEL
LIN {X 0,Y 386.91,Z 518.232,A -85,B 0,C 180,E1 -12305.306,E2 -12305.306} C_VEL
LIN {X 0,Y 385.451,Z 531.869,A -85,B 0,C 180,E1 -12306.222,E2 -12306.222} C_VEL
LIN {X 0,Y 383.796,Z 545.662,A -85,B 0,C 180,E1 -12307.385,E2 -12307.385} C_VEL
LIN {X 0,Y 382.114,Z 558.368,A -85,B 0,C 180,E1 -12308.701,E2 -12308.701} C_VEL
LIN {X 0,Y 380.635,Z 569.06,A -85,B 0,C 180,E1 -12310.027,E2 -12310.027} C_VEL
LIN {X 0,Y 379.153,Z 579.947,A -85,B 0,C 180,E1 -12311.633,E2 -12311.633} C_VEL
LIN {X 0,Y 377.711,Z 590.554,A -85,B 0,C 180,E1 -12313.516,E2 -12313.516} C_VEL
LIN {X 0,Y 376.515,Z 599.387,A -85,B 0,C 180,E1 -12315.405,E2 -12315.405} C_VEL
LIN {X 0,Y 375.632,Z 607.678,A -85,B 0,C 180,E1 -12317.575,E2 -12317.575} C_VEL
LIN {X 0,Y 374.977,Z 614.324,A -85,B 0,C 180,E1 -12319.744,E2 -12319.744} C_VEL
LIN {X 0,Y 374.69,Z 619.534,A -85,B 0,C 180,E1 -12321.914,E2 -12321.914} C_VEL
LIN {X 0,Y 374.559,Z 623.266,A -85,B 0,C 180,E1 -12323.965,E2 -12323.965} C_VEL
LIN {X 0,Y 374.519,Z 625.488,A -85,B 0,C 180,E1 -12325.696,E2 -12325.696} C_VEL
LIN {X 0,Y 374.5,Z 627.24,A -85,B 0,C 180,E1 -12327.85,E2 -12327.85} C_VEL
LIN {X 0,Y 374.587,Z 627.843,A -85,B 0,C 180,E1 -12330.001,E2 -12330.001} C_VEL
LIN {X 0,Y 374.5,Z 627.234,A -85,B 0,C 180,E1 -12332.151,E2 -12332.151} C_VEL
LIN {X 0,Y 374.518,Z 625.473,A -85,B 0,C 180,E1 -12334.305,E2 -12334.305} C_VEL
LIN {X 0,Y 374.562,Z 622.531,A -85,B 0,C 180,E1 -12336.465,E2 -12336.465} C_VEL
LIN {X 0,Y 374.727,Z 618.34,A -85,B 0,C 180,E1 -12338.63,E2 -12338.63} C_VEL
LIN {X 0,Y 375.114,Z 612.794,A -85,B 0,C 180,E1 -12340.799,E2 -12340.799} C_VEL
LIN {X 0,Y 375.865,Z 605.748,A -85,B 0,C 180,E1 -12342.967,E2 -12342.967} C_VEL
LIN {X 0,Y 376.666,Z 598.21,A -85,B 0,C 180,E1 -12344.866,E2 -12344.866} C_VEL
LIN {X 0,Y 377.821,Z 589.133,A -85,B 0,C 180,E1 -12346.758,E2 -12346.758} C_VEL
LIN {X 0,Y 379.376,Z 578.449,A -85,B 0,C 180,E1 -12348.601,E2 -12348.601} C_VEL
LIN {X 0,Y 380.883,Z 567.018,A -85,B 0,C 180,E1 -12350.242,E2 -12350.242} C_VEL
LIN {X 0,Y 382.563,Z 554.738,A -85,B 0,C 180,E1 -12351.699,E2 -12351.699} C_VEL
LIN {X 0,Y 384.351,Z 541.245,A -85,B 0,C 180,E1 -12353.008,E2 -12353.008} C_VEL
LIN {X 0,Y 385.98,Z 526.936,A -85,B 0,C 180,E1 -12354.128,E2 -12354.128} C_VEL
LIN {X 0,Y 387.471,Z 511.898,A -85,B 0,C 180,E1 -12355.044,E2 -12355.044} C_VEL
LIN {X 0,Y 388.592,Z 497.828,A -85,B 0,C 180,E1 -12355.687,E2 -12355.687} C_VEL
LIN {X 0,Y 389.544,Z 481.757,A -85,B 0,C 180,E1 -12356.197,E2 -12356.197} C_VEL
LIN {X 0,Y 392.458,Z 357.923,A -85,B 0,C 180,E1 -12358.514,E2 -12358.514} C_VEL
LIN {X 0,Y 391.79,Z 352.802,A -85,B 0,C 180,E1 -12358.671,E2 -12358.671} C_VEL
LIN {X 0,Y 386.942,Z 326.661,A -85,B 0,C 180,E1 -12359.603,E2 -12359.603} C_VEL
LIN {X 0,Y 385.165,Z 319.399,A -85,B 0,C 180,E1 -12359.904,E2 -12359.904} C_VEL
LIN {X 0,Y 383.179,Z 314.473,A -85,B 0,C 180,E1 -12360.208,E2 -12360.208} C_VEL
LIN {X 0,Y 379.451,Z 298.957,A -85,B 0,C 180,E1 -12363.544,E2 -12363.544} C_VEL
LIN {X 0,Y 375.98,Z 286.276,A -85,B 0,C 180,E1 -12366.455,E2 -12366.455} C_VEL
LIN {X 0,Y 375.988,Z 286.266,A -85,B 0,C 180,E1 -12369.971,E2 -12369.971} C_VEL
LIN {X 0,Y 375.931,Z 286.28,A -85,B 0,C 180,E1 -12373.767,E2 -12373.767} C_VEL
LIN {X 0,Y 375.936,Z 286.271,A -85,B 0,C 180,E1 -12376.811,E2 -12376.811} C_VEL
LIN {X 0,Y 375.964,Z 286.28,A -85,B 0,C 180,E1 -12380.538,E2 -12380.538} C_VEL
LIN {X 0,Y 375.967,Z 286.275,A -85,B 0,C 180,E1 -12383.496,E2 -12383.496} C_VEL
LIN {X 0,Y 375.964,Z 286.275,A -85,B 0,C 180,E1 -12385.889,E2 -12385.889} C_VEL
LIN {X 0,Y 375.966,Z 286.275,A -85,B 0,C 180,E1 -12389.688,E2 -12389.688} C_VEL
LIN {X 0,Y 375.938,Z 286.275,A -85,B 0,C 180,E1 -12393.342,E2 -12393.342} C_VEL
LIN {X 0,Y 375.982,Z 286.267,A -85,B 0,C 180,E1 -12396.887,E2 -12396.887} C_VEL
LIN {X 0,Y 376.002,Z 286.268,A -85,B 0,C 180,E1 -12400.34,E2 -12400.34} C_VEL
LIN {X 0,Y 376.034,Z 286.271,A -85,B 0,C 180,E1 -12403.719,E2 -12403.719} C_VEL
LIN {X 0,Y 376.108,Z 286.258,A -85,B 0,C 180,E1 -12407.042,E2 -12407.042} C_VEL
LIN {X 0,Y 376.117,Z 286.26,A -85,B 0,C 180,E1 -12410.319,E2 -12410.319} C_VEL
LIN {X 0,Y 376.203,Z 286.241,A -85,B 0,C 180,E1 -12413.564,E2 -12413.564} C_VEL
LIN {X 0,Y 376.342,Z 286.226,A -85,B 0,C 180,E1 -12417.86,E2 -12417.86} C_VEL
LIN {X 0,Y 376.347,Z 286.226,A -85,B 0,C 180,E1 -12422.141,E2 -12422.141} C_VEL
LIN {X 0,Y 376.194,Z 286.244,A -85,B 0,C 180,E1 -12426.451,E2 -12426.451} C_VEL
LIN {X 0,Y 376.114,Z 286.256,A -85,B 0,C 180,E1 -12429.682,E2 -12429.682} C_VEL
LIN {X 0,Y 376.095,Z 286.26,A -85,B 0,C 180,E1 -12433.658,E2 -12433.658} C_VEL
LIN {X 0,Y 375.987,Z 286.275,A -85,B 0,C 180,E1 -12437.577,E2 -12437.577} C_VEL
LIN {X 0,Y 375.983,Z 286.274,A -85,B 0,C 180,E1 -12440.832,E2 -12440.832} C_VEL
LIN {X 0,Y 375.938,Z 286.28,A -85,B 0,C 180,E1 -12444.285,E2 -12444.285} C_VEL
LIN {X 0,Y 375.913,Z 286.276,A -85,B 0,C 180,E1 -12446.66,E2 -12446.66} C_VEL
LIN {X 0,Y 375.916,Z 286.266,A -85,B 0,C 180,E1 -12449.084,E2 -12449.084} C_VEL
LIN {X 0,Y 375.956,Z 286.281,A -85,B 0,C 180,E1 -12451.562,E2 -12451.562} C_VEL
LIN {X 0,Y 375.951,Z 286.278,A -85,B 0,C 180,E1 -12455.416,E2 -12455.416} C_VEL
LIN {X 0,Y 375.935,Z 286.277,A -85,B 0,C 180,E1 -12458.262,E2 -12458.262} C_VEL
LIN {X 0,Y 375.912,Z 286.282,A -85,B 0,C 180,E1 -12461.596,E2 -12461.596} C_VEL
LIN {X 0,Y 375.874,Z 286.29,A -85,B 0,C 180,E1 -12465.277,E2 -12465.277} C_VEL
LIN {X 0,Y 375.911,Z 286.286,A -85,B 0,C 180,E1 -12469.128,E2 -12469.128} C_VEL
LIN {X 0,Y 375.952,Z 286.277,A -85,B 0,C 180,E1 -12471.909,E2 -12471.909} C_VEL
LIN {X 0,Y 375.977,Z 286.271,A -85,B 0,C 180,E1 -12475.334,E2 -12475.334} C_VEL
LIN {X 0,Y 375.959,Z 286.384,A -85,B 0,C 180,E1 -12478.32,E2 -12478.32} C_VEL
LIN {X 0,Y 377.066,Z 290.478,A -85,B 0,C 180,E1 -12479.348,E2 -12479.348} C_VEL
LIN {X 0,Y 386.773,Z 310.638,A -85,B 0,C 180,E1 -12480.629,E2 -12480.629} C_VEL
LIN {X 0,Y 392.92,Z 324.836,A -85,B 0,C 180,E1 -12481.429,E2 -12481.429} C_VEL
LIN {X 0,Y 390.978,Z 417.126,A -85,B 0,C 180,E1 -12483.154,E2 -12483.154} C_VEL
LIN {X 0,Y 389.971,Z 455.961,A -85,B 0,C 180,E1 -12483.905,E2 -12483.905} C_VEL
LIN {X 0,Y 389.232,Z 471.049,A -85,B 0,C 180,E1 -12484.401,E2 -12484.401} C_VEL
LIN {X 0,Y 388.376,Z 484.375,A -85,B 0,C 180,E1 -12485.022,E2 -12485.022} C_VEL
LIN {X 0,Y 387.148,Z 498.662,A -85,B 0,C 180,E1 -12485.892,E2 -12485.892} C_VEL
LIN {X 0,Y 385.691,Z 512.226,A -85,B 0,C 180,E1 -12486.935,E2 -12486.935} C_VEL
LIN {X 0,Y 383.941,Z 525.983,A -85,B 0,C 180,E1 -12488.242,E2 -12488.242} C_VEL
LIN {X 0,Y 382.326,Z 538.48,A -85,B 0,C 180,E1 -12489.711,E2 -12489.711} C_VEL
LIN {X 0,Y 380.871,Z 548.76,A -85,B 0,C 180,E1 -12491.16,E2 -12491.16} C_VEL
LIN {X 0,Y 379.484,Z 558.381,A -85,B 0,C 180,E1 -12492.763,E2 -12492.763} C_VEL
LIN {X 0,Y 378.077,Z 567.808,A -85,B 0,C 180,E1 -12494.639,E2 -12494.639} C_VEL
LIN {X 0,Y 377.089,Z 575.646,A -85,B 0,C 180,E1 -12496.528,E2 -12496.528} C_VEL
LIN {X 0,Y 376.046,Z 582.965,A -85,B 0,C 180,E1 -12498.682,E2 -12498.682} C_VEL
LIN {X 0,Y 375.405,Z 588.765,A -85,B 0,C 180,E1 -12500.843,E2 -12500.843} C_VEL
LIN {X 0,Y 375.061,Z 592.197,A -85,B 0,C 180,E1 -12502.462,E2 -12502.462} C_VEL
LIN {X 0,Y 374.81,Z 595.673,A -85,B 0,C 180,E1 -12504.62,E2 -12504.62} C_VEL
LIN {X 0,Y 374.61,Z 597.973,A -85,B 0,C 180,E1 -12506.773,E2 -12506.773} C_VEL
LIN {X 0,Y 374.594,Z 599.145,A -85,B 0,C 180,E1 -12508.924,E2 -12508.924} C_VEL
LIN {X 0,Y 374.594,Z 599.161,A -85,B 0,C 180,E1 -12511.075,E2 -12511.075} C_VEL
LIN {X 0,Y 374.609,Z 598.051,A -85,B 0,C 180,E1 -12513.226,E2 -12513.226} C_VEL
LIN {X 0,Y 374.703,Z 596.542,A -85,B 0,C 180,E1 -12514.757,E2 -12514.757} C_VEL
LIN {X 0,Y 374.159,Z 595.515,A -85,B 0,C 180,E1 -12515.642,E2 -12515.642} C_VEL
LIN {X 0,Y 371.513,Z 593.48,A -85,B 0,C 180,E1 -12517.078,E2 -12517.078} C_VEL
LIN {X 0,Y 369.287,Z 591.546,A -85,B 0,C 180,E1 -12518.225,E2 -12518.225} C_VEL
LIN {X 0,Y 368.413,Z 589.787,A -85,B 0,C 180,E1 -12519.096,E2 -12519.096} C_VEL
LIN {X 0,Y 368.387,Z 589.131,A -85,B 0,C 180,E1 -12519.386,E2 -12519.386} C_VEL
LIN {X 0,Y 369.036,Z 583.532,A -85,B 0,C 180,E1 -12521.534,E2 -12521.534} C_VEL
LIN {X 0,Y 370.095,Z 576.291,A -85,B 0,C 180,E1 -12523.731,E2 -12523.731} C_VEL
LIN {X 0,Y 371.166,Z 568.528,A -85,B 0,C 180,E1 -12525.653,E2 -12525.653} C_VEL
LIN {X 0,Y 372.627,Z 559.189,A -85,B 0,C 180,E1 -12527.564,E2 -12527.564} C_VEL
LIN {X 0,Y 374.057,Z 549.675,A -85,B 0,C 180,E1 -12529.195,E2 -12529.195} C_VEL
LIN {X 0,Y 375.735,Z 538.356,A -85,B 0,C 180,E1 -12530.817,E2 -12530.817} C_VEL
LIN {X 0,Y 377.492,Z 525.886,A -85,B 0,C 180,E1 -12532.292,E2 -12532.292} C_VEL
LIN {X 0,Y 379.055,Z 513.634,A -85,B 0,C 180,E1 -12533.492,E2 -12533.492} C_VEL
LIN {X 0,Y 380.57,Z 500.327,A -85,B 0,C 180,E1 -12534.551,E2 -12534.551} C_VEL
LIN {X 0,Y 381.847,Z 486.45,A -85,B 0,C 180,E1 -12535.428,E2 -12535.428} C_VEL
LIN {X 0,Y 382.925,Z 470.996,A -85,B 0,C 180,E1 -12536.171,E2 -12536.171} C_VEL
LIN {X 0,Y 383.638,Z 456.068,A -85,B 0,C 180,E1 -12536.668,E2 -12536.668} C_VEL
LIN {X 0,Y 384.955,Z 408.026,A -85,B 0,C 180,E1 -12537.597,E2 -12537.597} C_VEL
LIN {X 0,Y 386.762,Z 326.934,A -85,B 0,C 180,E1 -12539.135,E2 -12539.135} C_VEL
LIN {X 0,Y 378.319,Z 307.795,A -85,B 0,C 180,E1 -12540.27,E2 -12540.27} C_VEL
LIN {X 0,Y 369.766,Z 290.572,A -85,B 0,C 180,E1 -12541.462,E2 -12541.462} C_VEL
LIN {X 0,Y 368.905,Z 287.162,A -85,B 0,C 180,E1 -12542.373,E2 -12542.373} C_VEL
LIN {X 0,Y 368.921,Z 287.158,A -85,B 0,C 180,E1 -12544.999,E2 -12544.999} C_VEL
LIN {X 0,Y 368.874,Z 287.163,A -85,B 0,C 180,E1 -12548.633,E2 -12548.633} C_VEL
LIN {X 0,Y 368.856,Z 287.16,A -85,B 0,C 180,E1 -12552.005,E2 -12552.005} C_VEL
LIN {X 0,Y 368.871,Z 287.163,A -85,B 0,C 180,E1 -12555.174,E2 -12555.174} C_VEL
LIN {X 0,Y 368.858,Z 287.144,A -85,B 0,C 180,E1 -12558.174,E2 -12558.174} C_VEL
LIN {X 0,Y 368.872,Z 287.158,A -85,B 0,C 180,E1 -12561.366,E2 -12561.366} C_VEL
LIN {X 0,Y 368.928,Z 287.142,A -85,B 0,C 180,E1 -12565.145,E2 -12565.145} C_VEL
LIN {X 0,Y 368.894,Z 287.155,A -85,B 0,C 180,E1 -12569.043,E2 -12569.043} C_VEL
LIN {X 0,Y 368.904,Z 287.154,A -85,B 0,C 180,E1 -12571.557,E2 -12571.557} C_VEL
LIN {X 0,Y 368.917,Z 287.153,A -85,B 0,C 180,E1 -12574.013,E2 -12574.013} C_VEL
LIN {X 0,Y 368.893,Z 287.153,A -85,B 0,C 180,E1 -12577.602,E2 -12577.602} C_VEL
LIN {X 0,Y 368.898,Z 287.148,A -85,B 0,C 180,E1 -12581.103,E2 -12581.103} C_VEL
LIN {X 0,Y 368.932,Z 287.151,A -85,B 0,C 180,E1 -12584.532,E2 -12584.532} C_VEL
LIN {X 0,Y 369.056,Z 287.135,A -85,B 0,C 180,E1 -12586.79,E2 -12586.79} C_VEL
LIN {X 0,Y 369.058,Z 287.132,A -85,B 0,C 180,E1 -12590.131,E2 -12590.131} C_VEL
LIN {X 0,Y 369.151,Z 287.125,A -85,B 0,C 180,E1 -12593.441,E2 -12593.441} C_VEL
LIN {X 0,Y 369.306,Z 287.105,A -85,B 0,C 180,E1 -12597.819,E2 -12597.819} C_VEL
LIN {X 0,Y 369.302,Z 287.102,A -85,B 0,C 180,E1 -12602.181,E2 -12602.181} C_VEL
LIN {X 0,Y 369.159,Z 287.12,A -85,B 0,C 180,E1 -12606.559,E2 -12606.559} C_VEL
LIN {X 0,Y 369.061,Z 287.134,A -85,B 0,C 180,E1 -12609.868,E2 -12609.868} C_VEL
LIN {X 0,Y 369.036,Z 287.143,A -85,B 0,C 180,E1 -12613.772,E2 -12613.772} C_VEL
LIN {X 0,Y 369,Z 287.149,A -85,B 0,C 180,E1 -12617.768,E2 -12617.768} C_VEL
LIN {X 0,Y 368.927,Z 287.154,A -85,B 0,C 180,E1 -12621.22,E2 -12621.22} C_VEL
LIN {X 0,Y 368.933,Z 287.128,A -85,B 0,C 180,E1 -12624.777,E2 -12624.777} C_VEL
LIN {X 0,Y 368.915,Z 287.156,A -85,B 0,C 180,E1 -12628.441,E2 -12628.441} C_VEL
LIN {X 0,Y 368.908,Z 287.142,A -85,B 0,C 180,E1 -12630.987,E2 -12630.987} C_VEL
LIN {X 0,Y 368.935,Z 287.152,A -85,B 0,C 180,E1 -12634.854,E2 -12634.854} C_VEL
LIN {X 0,Y 368.908,Z 287.15,A -85,B 0,C 180,E1 -12638.641,E2 -12638.641} C_VEL
LIN {X 0,Y 368.88,Z 287.162,A -85,B 0,C 180,E1 -12642.01,E2 -12642.01} C_VEL
LIN {X 0,Y 368.878,Z 287.158,A -85,B 0,C 180,E1 -12645.176,E2 -12645.176} C_VEL
LIN {X 0,Y 368.881,Z 287.156,A -85,B 0,C 180,E1 -12648.178,E2 -12648.178} C_VEL
LIN {X 0,Y 368.906,Z 287.156,A -85,B 0,C 180,E1 -12651.36,E2 -12651.36} C_VEL
LIN {X 0,Y 368.924,Z 287.267,A -85,B 0,C 180,E1 -12652.989,E2 -12652.989} C_VEL
LIN {X 0,Y 372.595,Z 300.411,A -85,B 0,C 180,E1 -12656.092,E2 -12656.092} C_VEL
LIN {X 0,Y 376.032,Z 314.591,A -85,B 0,C 180,E1 -12659.181,E2 -12659.181} C_VEL
LIN {X 0,Y 379.888,Z 323.787,A -85,B 0,C 180,E1 -12659.721,E2 -12659.721} C_VEL
LIN {X 0,Y 384.28,Z 346.391,A -85,B 0,C 180,E1 -12660.574,E2 -12660.574} C_VEL
LIN {X 0,Y 386.224,Z 358.452,A -85,B 0,C 180,E1 -12660.986,E2 -12660.986} C_VEL
LIN {X 0,Y 383.403,Z 476.121,A -85,B 0,C 180,E1 -12663.204,E2 -12663.204} C_VEL
LIN {X 0,Y 382.684,Z 491.552,A -85,B 0,C 180,E1 -12663.628,E2 -12663.628} C_VEL
LIN {X 0,Y 381.545,Z 505.874,A -85,B 0,C 180,E1 -12664.205,E2 -12664.205} C_VEL
LIN {X 0,Y 380.17,Z 520.726,A -85,B 0,C 180,E1 -12665.03,E2 -12665.03} C_VEL
LIN {X 0,Y 378.537,Z 534.823,A -85,B 0,C 180,E1 -12666.038,E2 -12666.038} C_VEL
LIN {X 0,Y 376.852,Z 548.157,A -85,B 0,C 180,E1 -12667.234,E2 -12667.234} C_VEL
LIN {X 0,Y 374.925,Z 561.501,A -85,B 0,C 180,E1 -12668.704,E2 -12668.704} C_VEL
LIN {X 0,Y 373.144,Z 573.67,A -85,B 0,C 180,E1 -12670.343,E2 -12670.343} C_VEL
LIN {X 0,Y 371.664,Z 584.477,A -85,B 0,C 180,E1 -12672.105,E2 -12672.105} C_VEL
LIN {X 0,Y 370.226,Z 594.276,A -85,B 0,C 180,E1 -12674.023,E2 -12674.023} C_VEL
LIN {X 0,Y 369.078,Z 602.91,A -85,B 0,C 180,E1 -12676.074,E2 -12676.074} C_VEL
LIN {X 0,Y 368.451,Z 609.236,A -85,B 0,C 180,E1 -12677.889,E2 -12677.889} C_VEL
LIN {X 0,Y 367.816,Z 615.495,A -85,B 0,C 180,E1 -12680.098,E2 -12680.098} C_VEL
LIN {X 0,Y 367.561,Z 620.344,A -85,B 0,C 180,E1 -12682.309,E2 -12682.309} C_VEL
LIN {X 0,Y 367.419,Z 623.898,A -85,B 0,C 180,E1 -12684.512,E2 -12684.512} C_VEL
LIN {X 0,Y 367.378,Z 626.238,A -85,B 0,C 180,E1 -12686.71,E2 -12686.71} C_VEL
LIN {X 0,Y 367.482,Z 627.418,A -85,B 0,C 180,E1 -12688.905,E2 -12688.905} C_VEL
LIN {X 0,Y 367.482,Z 627.416,A -85,B 0,C 180,E1 -12691.096,E2 -12691.096} C_VEL
LIN {X 0,Y 367.378,Z 626.226,A -85,B 0,C 180,E1 -12693.291,E2 -12693.291} C_VEL
LIN {X 0,Y 367.417,Z 623.88,A -85,B 0,C 180,E1 -12695.489,E2 -12695.489} C_VEL
LIN {X 0,Y 367.56,Z 620.325,A -85,B 0,C 180,E1 -12697.692,E2 -12697.692} C_VEL
LIN {X 0,Y 367.813,Z 615.471,A -85,B 0,C 180,E1 -12699.903,E2 -12699.903} C_VEL
LIN {X 0,Y 368.451,Z 609.196,A -85,B 0,C 180,E1 -12702.112,E2 -12702.112} C_VEL
LIN {X 0,Y 369.271,Z 601.319,A -85,B 0,C 180,E1 -12704.325,E2 -12704.325} C_VEL
LIN {X 0,Y 370.414,Z 592.954,A -85,B 0,C 180,E1 -12706.252,E2 -12706.252} C_VEL
LIN {X 0,Y 371.891,Z 582.886,A -85,B 0,C 180,E1 -12708.169,E2 -12708.169} C_VEL
LIN {X 0,Y 373.35,Z 572.593,A -85,B 0,C 180,E1 -12709.807,E2 -12709.807} C_VEL
LIN {X 0,Y 375.078,Z 560.336,A -85,B 0,C 180,E1 -12711.432,E2 -12711.432} C_VEL
LIN {X 0,Y 376.996,Z 546.699,A -85,B 0,C 180,E1 -12712.903,E2 -12712.903} C_VEL
LIN {X 0,Y 378.749,Z 533.034,A -85,B 0,C 180,E1 -12714.094,E2 -12714.094} C_VEL
LIN {X 0,Y 380.289,Z 519.32,A -85,B 0,C 180,E1 -12715.052,E2 -12715.052} C_VEL
LIN {X 0,Y 381.619,Z 504.315,A -85,B 0,C 180,E1 -12715.865,E2 -12715.865} C_VEL
LIN {X 0,Y 382.836,Z 488.339,A -85,B 0,C 180,E1 -12716.472,E2 -12716.472} C_VEL
LIN {X 0,Y 383.503,Z 472.317,A -85,B 0,C 180,E1 -12716.863,E2 -12716.863} C_VEL
LIN {X 0,Y 386.189,Z 357.633,A -85,B 0,C 180,E1 -12719.02,E2 -12719.02} C_VEL
LIN {X 0,Y 380.975,Z 329.012,A -85,B 0,C 180,E1 -12720.058,E2 -12720.058} C_VEL
LIN {X 0,Y 379.355,Z 322.267,A -85,B 0,C 180,E1 -12720.342,E2 -12720.342} C_VEL
LIN {X 0,Y 375.92,Z 314.138,A -85,B 0,C 180,E1 -12720.857,E2 -12720.857} C_VEL
LIN {X 0,Y 372.119,Z 298.584,A -85,B 0,C 180,E1 -12724.307,E2 -12724.307} C_VEL
LIN {X 0,Y 368.903,Z 287.158,A -85,B 0,C 180,E1 -12727.064,E2 -12727.064} C_VEL
LIN {X 0,Y 368.91,Z 287.15,A -85,B 0,C 180,E1 -12730.371,E2 -12730.371} C_VEL
LIN {X 0,Y 368.884,Z 287.158,A -85,B 0,C 180,E1 -12733.616,E2 -12733.616} C_VEL
LIN {X 0,Y 368.888,Z 287.148,A -85,B 0,C 180,E1 -12736.696,E2 -12736.696} C_VEL
LIN {X 0,Y 368.914,Z 287.154,A -85,B 0,C 180,E1 -12739.644,E2 -12739.644} C_VEL
LIN {X 0,Y 368.904,Z 287.155,A -85,B 0,C 180,E1 -12743.145,E2 -12743.145} C_VEL
LIN {X 0,Y 368.9,Z 287.155,A -85,B 0,C 180,E1 -12746.462,E2 -12746.462} C_VEL
LIN {X 0,Y 368.933,Z 287.149,A -85,B 0,C 180,E1 -12749.047,E2 -12749.047} C_VEL
LIN {X 0,Y 368.879,Z 287.155,A -85,B 0,C 180,E1 -12752.79,E2 -12752.79} C_VEL
LIN {X 0,Y 368.932,Z 287.152,A -85,B 0,C 180,E1 -12756.119,E2 -12756.119} C_VEL
LIN {X 0,Y 368.941,Z 287.152,A -85,B 0,C 180,E1 -12759.947,E2 -12759.947} C_VEL
LIN {X 0,Y 368.981,Z 287.147,A -85,B 0,C 180,E1 -12763.399,E2 -12763.399} C_VEL
LIN {X 0,Y 369.063,Z 287.136,A -85,B 0,C 180,E1 -12766.791,E2 -12766.791} C_VEL
LIN {X 0,Y 369.067,Z 287.138,A -85,B 0,C 180,E1 -12770.132,E2 -12770.132} C_VEL
LIN {X 0,Y 369.164,Z 287.117,A -85,B 0,C 180,E1 -12773.441,E2 -12773.441} C_VEL
LIN {X 0,Y 369.306,Z 287.102,A -85,B 0,C 180,E1 -12777.819,E2 -12777.819} C_VEL
LIN {X 0,Y 369.31,Z 287.103,A -85,B 0,C 180,E1 -12782.181,E2 -12782.181} C_VEL
LIN {X 0,Y 369.158,Z 287.12,A -85,B 0,C 180,E1 -12786.559,E2 -12786.559} C_VEL
LIN {X 0,Y 369.065,Z 287.132,A -85,B 0,C 180,E1 -12789.868,E2 -12789.868} C_VEL
LIN {X 0,Y 369.042,Z 287.137,A -85,B 0,C 180,E1 -12793.772,E2 -12793.772} C_VEL
LIN {X 0,Y 368.958,Z 287.148,A -85,B 0,C 180,E1 -12797.745,E2 -12797.745} C_VEL
LIN {X 0,Y 368.913,Z 287.158,A -85,B 0,C 180,E1 -12801.221,E2 -12801.221} C_VEL
LIN {X 0,Y 368.912,Z 287.158,A -85,B 0,C 180,E1 -12803.873,E2 -12803.873} C_VEL
LIN {X 0,Y 368.86,Z 287.145,A -85,B 0,C 180,E1 -12807.212,E2 -12807.212} C_VEL
LIN {X 0,Y 368.895,Z 287.148,A -85,B 0,C 180,E1 -12809.692,E2 -12809.692} C_VEL
LIN {X 0,Y 368.899,Z 287.155,A -85,B 0,C 180,E1 -12813.042,E2 -12813.042} C_VEL
LIN {X 0,Y 368.913,Z 287.152,A -85,B 0,C 180,E1 -12816.197,E2 -12816.197} C_VEL
LIN {X 0,Y 368.874,Z 287.157,A -85,B 0,C 180,E1 -12818.957,E2 -12818.957} C_VEL
LIN {X 0,Y 368.856,Z 287.161,A -85,B 0,C 180,E1 -12822.004,E2 -12822.004} C_VEL
LIN {X 0,Y 368.829,Z 287.168,A -85,B 0,C 180,E1 -12825.167,E2 -12825.167} C_VEL
LIN {X 0,Y 368.841,Z 287.161,A -85,B 0,C 180,E1 -12828.171,E2 -12828.171} C_VEL
LIN {X 0,Y 368.876,Z 287.162,A -85,B 0,C 180,E1 -12831.366,E2 -12831.366} C_VEL
LIN {X 0,Y 368.932,Z 287.15,A -85,B 0,C 180,E1 -12835.145,E2 -12835.145} C_VEL
LIN {X 0,Y 368.944,Z 287.193,A -85,B 0,C 180,E1 -12837.766,E2 -12837.766} C_VEL
LIN {X 0,Y 369.788,Z 290.673,A -85,B 0,C 180,E1 -12838.673,E2 -12838.673} C_VEL
LIN {X 0,Y 379.009,Z 309.311,A -85,B 0,C 180,E1 -12839.93,E2 -12839.93} C_VEL
LIN {X 0,Y 386.708,Z 326.961,A -85,B 0,C 180,E1 -12840.965,E2 -12840.965} C_VEL
LIN {X 0,Y 384.655,Z 417.636,A -85,B 0,C 180,E1 -12842.681,E2 -12842.681} C_VEL
LIN {X 0,Y 383.618,Z 456.247,A -85,B 0,C 180,E1 -12843.44,E2 -12843.44} C_VEL
LIN {X 0,Y 382.842,Z 471.436,A -85,B 0,C 180,E1 -12843.947,E2 -12843.947} C_VEL
LIN {X 0,Y 381.928,Z 485.194,A -85,B 0,C 180,E1 -12844.602,E2 -12844.602} C_VEL
LIN {X 0,Y 380.69,Z 498.939,A -85,B 0,C 180,E1 -12845.456,E2 -12845.456} C_VEL
LIN {X 0,Y 379.174,Z 512.502,A -85,B 0,C 180,E1 -12846.515,E2 -12846.515} C_VEL
LIN {X 0,Y 377.367,Z 526.258,A -85,B 0,C 180,E1 -12847.843,E2 -12847.843} C_VEL
LIN {X 0,Y 375.691,Z 538.37,A -85,B 0,C 180,E1 -12849.284,E2 -12849.284} C_VEL
LIN {X 0,Y 374.125,Z 549.035,A -85,B 0,C 180,E1 -12850.807,E2 -12850.807} C_VEL
LIN {X 0,Y 372.696,Z 558.655,A -85,B 0,C 180,E1 -12852.439,E2 -12852.439} C_VEL
LIN {X 0,Y 371.197,Z 568.083,A -85,B 0,C 180,E1 -12854.347,E2 -12854.347} C_VEL
LIN {X 0,Y 370.157,Z 575.919,A -85,B 0,C 180,E1 -12856.27,E2 -12856.27} C_VEL
LIN {X 0,Y 369.064,Z 583.238,A -85,B 0,C 180,E1 -12858.465,E2 -12858.465} C_VEL
LIN {X 0,Y 368.395,Z 589.037,A -85,B 0,C 180,E1 -12860.667,E2 -12860.667} C_VEL
LIN {X 0,Y 368.006,Z 592.47,A -85,B 0,C 180,E1 -12862.317,E2 -12862.317} C_VEL
LIN {X 0,Y 367.736,Z 595.944,A -85,B 0,C 180,E1 -12864.516,E2 -12864.516} C_VEL
LIN {X 0,Y 367.52,Z 598.244,A -85,B 0,C 180,E1 -12866.711,E2 -12866.711} C_VEL
LIN {X 0,Y 367.513,Z 599.415,A -85,B 0,C 180,E1 -12868.904,E2 -12868.904} C_VEL
LIN {X 0,Y 367.513,Z 599.43,A -85,B 0,C 180,E1 -12871.095,E2 -12871.095} C_VEL
LIN {X 0,Y 367.519,Z 598.321,A -85,B 0,C 180,E1 -12873.288,E2 -12873.288} C_VEL
LIN {X 0,Y 367.732,Z 596.081,A -85,B 0,C 180,E1 -12875.483,E2 -12875.483} C_VEL
LIN {X 0,Y 367.993,Z 592.662,A -85,B 0,C 180,E1 -12877.682,E2 -12877.682} C_VEL
LIN {X 0,Y 368.387,Z 589.131,A -85,B 0,C 180,E1 -12879.386,E2 -12879.386} C_VEL
LIN {X 0,Y 367.939,Z 587.129,A -85,B 0,C 180,E1 -12880.248,E2 -12880.248} C_VEL
LIN {X 0,Y 365.581,Z 583.662,A -85,B 0,C 180,E1 -12881.652,E2 -12881.652} C_VEL
LIN {X 0,Y 363.346,Z 579.772,A -85,B 0,C 180,E1 -12883.043,E2 -12883.043} C_VEL
LIN {X 0,Y 363.092,Z 577.022,A -85,B 0,C 180,E1 -12883.869,E2 -12883.869} C_VEL
LIN {X 0,Y 364.132,Z 570.017,A -85,B 0,C 180,E1 -12885.676,E2 -12885.676} C_VEL
LIN {X 0,Y 365.582,Z 560.932,A -85,B 0,C 180,E1 -12887.624,E2 -12887.624} C_VEL
LIN {X 0,Y 367.101,Z 551.667,A -85,B 0,C 180,E1 -12889.283,E2 -12889.283} C_VEL
LIN {X 0,Y 368.784,Z 540.475,A -85,B 0,C 180,E1 -12890.964,E2 -12890.964} C_VEL
LIN {X 0,Y 370.546,Z 528.604,A -85,B 0,C 180,E1 -12892.439,E2 -12892.439} C_VEL
LIN {X 0,Y 372.373,Z 515.353,A -85,B 0,C 180,E1 -12893.792,E2 -12893.792} C_VEL
LIN {X 0,Y 373.916,Z 502.354,A -85,B 0,C 180,E1 -12894.869,E2 -12894.869} C_VEL
LIN {X 0,Y 375.27,Z 488.518,A -85,B 0,C 180,E1 -12895.787,E2 -12895.787} C_VEL
LIN {X 0,Y 376.414,Z 473.627,A -85,B 0,C 180,E1 -12896.542,E2 -12896.542} C_VEL
LIN {X 0,Y 377.241,Z 458.596,A -85,B 0,C 180,E1 -12897.082,E2 -12897.082} C_VEL
LIN {X 0,Y 377.902,Z 438.642,A -85,B 0,C 180,E1 -12897.518,E2 -12897.518} C_VEL
LIN {X 0,Y 380.421,Z 336.421,A -85,B 0,C 180,E1 -12899.472,E2 -12899.472} C_VEL
LIN {X 0,Y 380.539,Z 328.815,A -85,B 0,C 180,E1 -12899.624,E2 -12899.624} C_VEL
LIN {X 0,Y 372.757,Z 311.288,A -85,B 0,C 180,E1 -12900.698,E2 -12900.698} C_VEL
LIN {X 0,Y 364.1,Z 293.979,A -85,B 0,C 180,E1 -12901.912,E2 -12901.912} C_VEL
LIN {X 0,Y 362.616,Z 290.906,A -85,B 0,C 180,E1 -12902.148,E2 -12902.148} C_VEL
LIN {X 0,Y 361.88,Z 288.033,A -85,B 0,C 180,E1 -12902.941,E2 -12902.941} C_VEL
LIN {X 0,Y 361.862,Z 288.031,A -85,B 0,C 180,E1 -12905.637,E2 -12905.637} C_VEL
LIN {X 0,Y 361.824,Z 288.043,A -85,B 0,C 180,E1 -12909.017,E2 -12909.017} C_VEL
LIN {X 0,Y 361.827,Z 288.027,A -85,B 0,C 180,E1 -12912.83,E2 -12912.83} C_VEL
LIN {X 0,Y 361.812,Z 288.04,A -85,B 0,C 180,E1 -12915.947,E2 -12915.947} C_VEL
LIN {X 0,Y 361.808,Z 288.033,A -85,B 0,C 180,E1 -12919.249,E2 -12919.249} C_VEL
LIN {X 0,Y 361.857,Z 288.012,A -85,B 0,C 180,E1 -12922.981,E2 -12922.981} C_VEL
LIN {X 0,Y 361.855,Z 288.037,A -85,B 0,C 180,E1 -12926.631,E2 -12926.631} C_VEL
LIN {X 0,Y 361.844,Z 288.033,A -85,B 0,C 180,E1 -12929.669,E2 -12929.669} C_VEL
